LIN {X 0,Y 573.239,Z 232.081,A -85,B 0,C 180,E1 -2291.594,E2 -2291.594} C_VEL
LIN {X 0,Y 573.228,Z 232.079,A -85,B 0,C 180,E1 -2294.334,E2 -2294.334} C_VEL
LIN {X 0,Y 573.226,Z 232.083,A -85,B 0,C 180,E1 -2297.36,E2 -2297.36} C_VEL
LIN {X 0,Y 573.227,Z 232.083,A -85,B 0,C 180,E1 -2300.391,E2 -2300.391} C_VEL
LIN {X 0,Y 573.23,Z 232.078,A -85,B 0,C 180,E1 -2303.076,E2 -2303.076} C_VEL
LIN {X 0,Y 573.267,Z 232.08,A -85,B 0,C 180,E1 -2305.671,E2 -2305.671} C_VEL
LIN {X 0,Y 573.251,Z 232.076,A -85,B 0,C 180,E1 -2308.185,E2 -2308.185} C_VEL
LIN {X 0,Y 573.258,Z 232.079,A -85,B 0,C 180,E1 -2310.634,E2 -2310.634} C_VEL
LIN {X 0,Y 573.212,Z 232.08,A -85,B 0,C 180,E1 -2313.513,E2 -2313.513} C_VEL
LIN {X 0,Y 573.208,Z 232.086,A -85,B 0,C 180,E1 -2316.133,E2 -2316.133} C_VEL
LIN {X 0,Y 573.254,Z 232.075,A -85,B 0,C 180,E1 -2318.709,E2 -2318.709} C_VEL
LIN {X 0,Y 573.225,Z 232.083,A -85,B 0,C 180,E1 -2321.411,E2 -2321.411} C_VEL
LIN {X 0,Y 573.244,Z 232.077,A -85,B 0,C 180,E1 -2323.621,E2 -2323.621} C_VEL
LIN {X 0,Y 573.259,Z 232.076,A -85,B 0,C 180,E1 -2325.807,E2 -2325.807} C_VEL
LIN {X 0,Y 573.265,Z 232.074,A -85,B 0,C 180,E1 -2328.746,E2 -2328.746} C_VEL
LIN {X 0,Y 573.243,Z 232.082,A -85,B 0,C 180,E1 -2331.54,E2 -2331.54} C_VEL
LIN {X 0,Y 573.238,Z 232.078,A -85,B 0,C 180,E1 -2333.665,E2 -2333.665} C_VEL
LIN {X 0,Y 573.226,Z 232.079,A -85,B 0,C 180,E1 -2335.781,E2 -2335.781} C_VEL
LIN {X 0,Y 573.311,Z 232.071,A -85,B 0,C 180,E1 -2337.892,E2 -2337.892} C_VEL
LIN {X 0,Y 573.318,Z 232.068,A -85,B 0,C 180,E1 -2340.702,E2 -2340.702} C_VEL
LIN {X 0,Y 573.216,Z 232.086,A -85,B 0,C 180,E1 -2343.515,E2 -2343.515} C_VEL
LIN {X 0,Y 573.281,Z 232.073,A -85,B 0,C 180,E1 -2345.628,E2 -2345.628} C_VEL
LIN {X 0,Y 573.269,Z 232.073,A -85,B 0,C 180,E1 -2347.75,E2 -2347.75} C_VEL
LIN {X 0,Y 573.267,Z 232.077,A -85,B 0,C 180,E1 -2350.597,E2 -2350.597} C_VEL
LIN {X 0,Y 573.264,Z 232.074,A -85,B 0,C 180,E1 -2352.749,E2 -2352.749} C_VEL
LIN {X 0,Y 573.227,Z 232.08,A -85,B 0,C 180,E1 -2354.92,E2 -2354.92} C_VEL
LIN {X 0,Y 573.216,Z 232.08,A -85,B 0,C 180,E1 -2357.85,E2 -2357.85} C_VEL
LIN {X 0,Y 573.238,Z 232.078,A -85,B 0,C 180,E1 -2360.077,E2 -2360.077} C_VEL
LIN {X 0,Y 573.236,Z 232.084,A -85,B 0,C 180,E1 -2362.338,E2 -2362.338} C_VEL
LIN {X 0,Y 573.25,Z 232.076,A -85,B 0,C 180,E1 -2364.37,E2 -2364.37} C_VEL
LIN {X 0,Y 572.626,Z 232.154,A -85,B 0,C 180,E1 -2364.956,E2 -2364.956} C_VEL
LIN {X 0,Y 569.79,Z 232.514,A -85,B 0,C 180,E1 -2365.907,E2 -2365.907} C_VEL
LIN {X 0,Y 567.357,Z 232.819,A -85,B 0,C 180,E1 -2366.673,E2 -2366.673} C_VEL
LIN {X 0,Y 566.295,Z 232.949,A -85,B 0,C 180,E1 -2367.264,E2 -2367.264} C_VEL
LIN {X 0,Y 566.201,Z 232.958,A -85,B 0,C 180,E1 -2367.464,E2 -2367.464} C_VEL
LIN {X 0,Y 566.165,Z 232.959,A -85,B 0,C 180,E1 -2369.771,E2 -2369.771} C_VEL
LIN {X 0,Y 566.201,Z 232.96,A -85,B 0,C 180,E1 -2372.429,E2 -2372.429} C_VEL
LIN {X 0,Y 566.171,Z 232.957,A -85,B 0,C 180,E1 -2374.988,E2 -2374.988} C_VEL
LIN {X 0,Y 566.194,Z 232.958,A -85,B 0,C 180,E1 -2377.461,E2 -2377.461} C_VEL
LIN {X 0,Y 566.209,Z 232.953,A -85,B 0,C 180,E1 -2380.199,E2 -2380.199} C_VEL
LIN {X 0,Y 566.19,Z 232.96,A -85,B 0,C 180,E1 -2383.056,E2 -2383.056} C_VEL
LIN {X 0,Y 566.147,Z 232.965,A -85,B 0,C 180,E1 -2386.055,E2 -2386.055} C_VEL
LIN {X 0,Y 566.158,Z 232.959,A -85,B 0,C 180,E1 -2388.859,E2 -2388.859} C_VEL
LIN {X 0,Y 566.212,Z 232.959,A -85,B 0,C 180,E1 -2391.442,E2 -2391.442} C_VEL
LIN {X 0,Y 566.142,Z 232.963,A -85,B 0,C 180,E1 -2394.306,E2 -2394.306} C_VEL
LIN {X 0,Y 566.181,Z 233.754,A -85,B 0,C 180,E1 -2395.18,E2 -2395.18} C_VEL
LIN {X 0,Y 566.128,Z 237.923,A -85,B 0,C 180,E1 -2397.737,E2 -2397.737} C_VEL
LIN {X 0,Y 566.072,Z 242.199,A -85,B 0,C 180,E1 -2400.352,E2 -2400.352} C_VEL
LIN {X 0,Y 566.044,Z 246.038,A -85,B 0,C 180,E1 -2402.652,E2 -2402.652} C_VEL
LIN {X 0,Y 566.044,Z 250.095,A -85,B 0,C 180,E1 -2405.03,E2 -2405.03} C_VEL
LIN {X 0,Y 565.985,Z 254.135,A -85,B 0,C 180,E1 -2407.36,E2 -2407.36} C_VEL
LIN {X 0,Y 565.954,Z 258.174,A -85,B 0,C 180,E1 -2409.653,E2 -2409.653} C_VEL
LIN {X 0,Y 565.908,Z 262.249,A -85,B 0,C 180,E1 -2411.912,E2 -2411.912} C_VEL
LIN {X 0,Y 565.89,Z 266.396,A -85,B 0,C 180,E1 -2414.144,E2 -2414.144} C_VEL
LIN {X 0,Y 565.905,Z 270.544,A -85,B 0,C 180,E1 -2416.352,E2 -2416.352} C_VEL
LIN {X 0,Y 565.903,Z 272.531,A -85,B 0,C 180,E1 -2417.402,E2 -2417.402} C_VEL
LIN {X 0,Y 566.906,Z 280.366,A -85,B 0,C 180,E1 -2417.607,E2 -2417.607} C_VEL
LIN {X 0,Y 566.754,Z 293.781,A -85,B 0,C 180,E1 -2418.012,E2 -2418.012} C_VEL
LIN {X 0,Y 566.661,Z 306.298,A -85,B 0,C 180,E1 -2418.554,E2 -2418.554} C_VEL
LIN {X 0,Y 566.529,Z 317.551,A -85,B 0,C 180,E1 -2419.191,E2 -2419.191} C_VEL
LIN {X 0,Y 566.337,Z 328.843,A -85,B 0,C 180,E1 -2419.995,E2 -2419.995} C_VEL
LIN {X 0,Y 566.238,Z 338.89,A -85,B 0,C 180,E1 -2420.895,E2 -2420.895} C_VEL
LIN {X 0,Y 566.113,Z 348.591,A -85,B 0,C 180,E1 -2421.972,E2 -2421.972} C_VEL
LIN {X 0,Y 566.05,Z 355.159,A -85,B 0,C 180,E1 -2422.868,E2 -2422.868} C_VEL
LIN {X 0,Y 566.003,Z 361.628,A -85,B 0,C 180,E1 -2423.942,E2 -2423.942} C_VEL
LIN {X 0,Y 565.878,Z 366.765,A -85,B 0,C 180,E1 -2425.013,E2 -2425.013} C_VEL
LIN {X 0,Y 565.926,Z 370.754,A -85,B 0,C 180,E1 -2426.084,E2 -2426.084} C_VEL
LIN {X 0,Y 565.878,Z 373.702,A -85,B 0,C 180,E1 -2427.153,E2 -2427.153} C_VEL
LIN {X 0,Y 565.839,Z 375.128,A -85,B 0,C 180,E1 -2427.865,E2 -2427.865} C_VEL
LIN {X 0,Y 565.841,Z 376.756,A -85,B 0,C 180,E1 -2429.288,E2 -2429.288} C_VEL
LIN {X 0,Y 565.839,Z 376.996,A -85,B 0,C 180,E1 -2430,E2 -2430} C_VEL
LIN {X 0,Y 565.841,Z 376.815,A -85,B 0,C 180,E1 -2430.712,E2 -2430.712} C_VEL
LIN {X 0,Y 565.838,Z 375.268,A -85,B 0,C 180,E1 -2432.136,E2 -2432.136} C_VEL
LIN {X 0,Y 565.879,Z 373.907,A -85,B 0,C 180,E1 -2432.848,E2 -2432.848} C_VEL
LIN {X 0,Y 565.926,Z 371.029,A -85,B 0,C 180,E1 -2433.917,E2 -2433.917} C_VEL
LIN {X 0,Y 565.878,Z 367.129,A -85,B 0,C 180,E1 -2434.988,E2 -2434.988} C_VEL
LIN {X 0,Y 565.99,Z 362.096,A -85,B 0,C 180,E1 -2436.059,E2 -2436.059} C_VEL
LIN {X 0,Y 566.031,Z 355.771,A -85,B 0,C 180,E1 -2437.133,E2 -2437.133} C_VEL
LIN {X 0,Y 566.128,Z 347.849,A -85,B 0,C 180,E1 -2438.208,E2 -2438.208} C_VEL
LIN {X 0,Y 566.249,Z 337.997,A -85,B 0,C 180,E1 -2439.285,E2 -2439.285} C_VEL
LIN {X 0,Y 566.405,Z 327.678,A -85,B 0,C 180,E1 -2440.184,E2 -2440.184} C_VEL
LIN {X 0,Y 566.502,Z 316.393,A -85,B 0,C 180,E1 -2440.973,E2 -2440.973} C_VEL
LIN {X 0,Y 566.692,Z 305.185,A -85,B 0,C 180,E1 -2441.592,E2 -2441.592} C_VEL
LIN {X 0,Y 566.791,Z 292.591,A -85,B 0,C 180,E1 -2442.119,E2 -2442.119} C_VEL
LIN {X 0,Y 566.935,Z 279.413,A -85,B 0,C 180,E1 -2442.507,E2 -2442.507} C_VEL
LIN {X 0,Y 565.906,Z 272.529,A -85,B 0,C 180,E1 -2442.689,E2 -2442.689} C_VEL
LIN {X 0,Y 565.918,Z 267.947,A -85,B 0,C 180,E1 -2445.117,E2 -2445.117} C_VEL
LIN {X 0,Y 565.923,Z 263.798,A -85,B 0,C 180,E1 -2447.341,E2 -2447.341} C_VEL
LIN {X 0,Y 565.942,Z 259.671,A -85,B 0,C 180,E1 -2449.59,E2 -2449.59} C_VEL
LIN {X 0,Y 565.983,Z 255.624,A -85,B 0,C 180,E1 -2451.871,E2 -2451.871} C_VEL
LIN {X 0,Y 565.981,Z 251.584,A -85,B 0,C 180,E1 -2454.191,E2 -2454.191} C_VEL
LIN {X 0,Y 566.025,Z 247.439,A -85,B 0,C 180,E1 -2456.622,E2 -2456.622} C_VEL
LIN {X 0,Y 566.094,Z 243.487,A -85,B 0,C 180,E1 -2458.959,E2 -2458.959} C_VEL
LIN {X 0,Y 566.094,Z 239.426,A -85,B 0,C 180,E1 -2461.428,E2 -2461.428} C_VEL
LIN {X 0,Y 566.153,Z 235.297,A -85,B 0,C 180,E1 -2463.96,E2 -2463.96} C_VEL
LIN {X 0,Y 566.16,Z 233.635,A -85,B 0,C 180,E1 -2464.986,E2 -2464.986} C_VEL
LIN {X 0,Y 566.143,Z 232.963,A -85,B 0,C 180,E1 -2465.694,E2 -2465.694} C_VEL
LIN {X 0,Y 566.214,Z 232.958,A -85,B 0,C 180,E1 -2468.558,E2 -2468.558} C_VEL
LIN {X 0,Y 566.168,Z 232.958,A -85,B 0,C 180,E1 -2471.14,E2 -2471.14} C_VEL
LIN {X 0,Y 566.149,Z 232.965,A -85,B 0,C 180,E1 -2474.041,E2 -2474.041} C_VEL
LIN {X 0,Y 566.196,Z 232.96,A -85,B 0,C 180,E1 -2477.084,E2 -2477.084} C_VEL
LIN {X 0,Y 566.217,Z 232.955,A -85,B 0,C 180,E1 -2480.314,E2 -2480.314} C_VEL
LIN {X 0,Y 566.203,Z 232.953,A -85,B 0,C 180,E1 -2483.43,E2 -2483.43} C_VEL
LIN {X 0,Y 566.199,Z 232.956,A -85,B 0,C 180,E1 -2486.268,E2 -2486.268} C_VEL
LIN {X 0,Y 566.183,Z 232.96,A -85,B 0,C 180,E1 -2488.926,E2 -2488.926} C_VEL
LIN {X 0,Y 566.196,Z 232.955,A -85,B 0,C 180,E1 -2491.856,E2 -2491.856} C_VEL
LIN {X 0,Y 566.218,Z 232.958,A -85,B 0,C 180,E1 -2494.251,E2 -2494.251} C_VEL
LIN {X 0,Y 566.173,Z 232.958,A -85,B 0,C 180,E1 -2496.719,E2 -2496.719} C_VEL
LIN {X 0,Y 566.208,Z 232.958,A -85,B 0,C 180,E1 -2499.663,E2 -2499.663} C_VEL
LIN {X 0,Y 566.174,Z 232.957,A -85,B 0,C 180,E1 -2501.921,E2 -2501.921} C_VEL
LIN {X 0,Y 566.188,Z 232.96,A -85,B 0,C 180,E1 -2504.89,E2 -2504.89} C_VEL
LIN {X 0,Y 566.241,Z 232.953,A -85,B 0,C 180,E1 -2507.819,E2 -2507.819} C_VEL
LIN {X 0,Y 566.212,Z 232.953,A -85,B 0,C 180,E1 -2510.714,E2 -2510.714} C_VEL
LIN {X 0,Y 566.22,Z 232.958,A -85,B 0,C 180,E1 -2513.205,E2 -2513.205} C_VEL
LIN {X 0,Y 566.265,Z 232.952,A -85,B 0,C 180,E1 -2515.016,E2 -2515.016} C_VEL
LIN {X 0,Y 566.264,Z 232.948,A -85,B 0,C 180,E1 -2517.866,E2 -2517.866} C_VEL
LIN {X 0,Y 566.301,Z 232.942,A -85,B 0,C 180,E1 -2520.711,E2 -2520.711} C_VEL
LIN {X 0,Y 566.275,Z 232.946,A -85,B 0,C 180,E1 -2522.846,E2 -2522.846} C_VEL
LIN {X 0,Y 566.258,Z 232.948,A -85,B 0,C 180,E1 -2525.698,E2 -2525.698} C_VEL
LIN {X 0,Y 566.197,Z 232.961,A -85,B 0,C 180,E1 -2528.566,E2 -2528.566} C_VEL
LIN {X 0,Y 566.197,Z 232.955,A -85,B 0,C 180,E1 -2531.455,E2 -2531.455} C_VEL
LIN {X 0,Y 566.226,Z 232.951,A -85,B 0,C 180,E1 -2534.501,E2 -2534.501} C_VEL
LIN {X 0,Y 566.203,Z 232.959,A -85,B 0,C 180,E1 -2537.332,E2 -2537.332} C_VEL
LIN {X 0,Y 566.211,Z 232.957,A -85,B 0,C 180,E1 -2540.337,E2 -2540.337} C_VEL
LIN {X 0,Y 566.168,Z 232.958,A -85,B 0,C 180,E1 -2543.28,E2 -2543.28} C_VEL
LIN {X 0,Y 566.189,Z 232.963,A -85,B 0,C 180,E1 -2545.75,E2 -2545.75} C_VEL
LIN {X 0,Y 566.188,Z 232.956,A -85,B 0,C 180,E1 -2548.198,E2 -2548.198} C_VEL
LIN {X 0,Y 566.192,Z 232.96,A -85,B 0,C 180,E1 -2551.076,E2 -2551.076} C_VEL
LIN {X 0,Y 566.215,Z 232.953,A -85,B 0,C 180,E1 -2553.734,E2 -2553.734} C_VEL
LIN {X 0,Y 566.183,Z 232.957,A -85,B 0,C 180,E1 -2556.571,E2 -2556.571} C_VEL
LIN {X 0,Y 566.206,Z 232.957,A -85,B 0,C 180,E1 -2559.684,E2 -2559.684} C_VEL
LIN {X 0,Y 566.175,Z 232.957,A -85,B 0,C 180,E1 -2562.091,E2 -2562.091} C_VEL
LIN {X 0,Y 566.167,Z 232.96,A -85,B 0,C 180,E1 -2565.037,E2 -2565.037} C_VEL
LIN {X 0,Y 566.192,Z 232.962,A -85,B 0,C 180,E1 -2567.91,E2 -2567.91} C_VEL
LIN {X 0,Y 566.212,Z 232.954,A -85,B 0,C 180,E1 -2570.726,E2 -2570.726} C_VEL
LIN {X 0,Y 566.222,Z 233.113,A -85,B 0,C 180,E1 -2573.638,E2 -2573.638} C_VEL
LIN {X 0,Y 566.512,Z 236.983,A -85,B 0,C 180,E1 -2575.203,E2 -2575.203} C_VEL
LIN {X 0,Y 566.453,Z 243.602,A -85,B 0,C 180,E1 -2577.757,E2 -2577.757} C_VEL
LIN {X 0,Y 566.335,Z 251.568,A -85,B 0,C 180,E1 -2580.68,E2 -2580.68} C_VEL
LIN {X 0,Y 566.252,Z 259.349,A -85,B 0,C 180,E1 -2583.46,E2 -2583.46} C_VEL
LIN {X 0,Y 566.223,Z 267.275,A -85,B 0,C 180,E1 -2586.209,E2 -2586.209} C_VEL
LIN {X 0,Y 566.155,Z 275.17,A -85,B 0,C 180,E1 -2588.9,E2 -2588.9} C_VEL
LIN {X 0,Y 566.088,Z 283.03,A -85,B 0,C 180,E1 -2591.543,E2 -2591.543} C_VEL
LIN {X 0,Y 566.028,Z 291.935,A -85,B 0,C 180,E1 -2594.517,E2 -2594.517} C_VEL
LIN {X 0,Y 565.98,Z 300.491,A -85,B 0,C 180,E1 -2597.335,E2 -2597.335} C_VEL
LIN {X 0,Y 566.952,Z 307.503,A -85,B 0,C 180,E1 -2597.494,E2 -2597.494} C_VEL
LIN {X 0,Y 566.827,Z 319.872,A -85,B 0,C 180,E1 -2597.832,E2 -2597.832} C_VEL
LIN {X 0,Y 566.645,Z 332.902,A -85,B 0,C 180,E1 -2598.346,E2 -2598.346} C_VEL
LIN {X 0,Y 566.526,Z 344.488,A -85,B 0,C 180,E1 -2598.955,E2 -2598.955} C_VEL
LIN {X 0,Y 566.438,Z 355.922,A -85,B 0,C 180,E1 -2599.726,E2 -2599.726} C_VEL
LIN {X 0,Y 566.282,Z 365.599,A -85,B 0,C 180,E1 -2600.535,E2 -2600.535} C_VEL
LIN {X 0,Y 566.181,Z 374.412,A -85,B 0,C 180,E1 -2601.433,E2 -2601.433} C_VEL
LIN {X 0,Y 566.056,Z 383.001,A -85,B 0,C 180,E1 -2602.509,E2 -2602.509} C_VEL
LIN {X 0,Y 565.965,Z 389.868,A -85,B 0,C 180,E1 -2603.583,E2 -2603.583} C_VEL
LIN {X 0,Y 565.937,Z 395.365,A -85,B 0,C 180,E1 -2604.656,E2 -2604.656} C_VEL
LIN {X 0,Y 565.959,Z 399.677,A -85,B 0,C 180,E1 -2605.727,E2 -2605.727} C_VEL
LIN {X 0,Y 565.927,Z 401.957,A -85,B 0,C 180,E1 -2606.44,E2 -2606.44} C_VEL
LIN {X 0,Y 565.878,Z 403.808,A -85,B 0,C 180,E1 -2607.152,E2 -2607.152} C_VEL
LIN {X 0,Y 565.846,Z 406.185,A -85,B 0,C 180,E1 -2608.577,E2 -2608.577} C_VEL
LIN {X 0,Y 565.839,Z 407,A -85,B 0,C 180,E1 -2610,E2 -2610} C_VEL
LIN {X 0,Y 565.846,Z 406.186,A -85,B 0,C 180,E1 -2611.423,E2 -2611.423} C_VEL
LIN {X 0,Y 565.878,Z 403.81,A -85,B 0,C 180,E1 -2612.847,E2 -2612.847} C_VEL
LIN {X 0,Y 565.926,Z 400.896,A -85,B 0,C 180,E1 -2613.916,E2 -2613.916} C_VEL
LIN {X 0,Y 565.878,Z 396.949,A -85,B 0,C 180,E1 -2614.987,E2 -2614.987} C_VEL
LIN {X 0,Y 566.002,Z 391.867,A -85,B 0,C 180,E1 -2616.058,E2 -2616.058} C_VEL
LIN {X 0,Y 566.04,Z 385.468,A -85,B 0,C 180,E1 -2617.132,E2 -2617.132} C_VEL
LIN {X 0,Y 566.134,Z 377.478,A -85,B 0,C 180,E1 -2618.208,E2 -2618.208} C_VEL
LIN {X 0,Y 566.229,Z 369.335,A -85,B 0,C 180,E1 -2619.105,E2 -2619.105} C_VEL
LIN {X 0,Y 566.339,Z 359.4,A -85,B 0,C 180,E1 -2620.005,E2 -2620.005} C_VEL
LIN {X 0,Y 566.471,Z 348.335,A -85,B 0,C 180,E1 -2620.806,E2 -2620.806} C_VEL
LIN {X 0,Y 566.608,Z 335.946,A -85,B 0,C 180,E1 -2621.51,E2 -2621.51} C_VEL
LIN {X 0,Y 566.742,Z 323.768,A -85,B 0,C 180,E1 -2622.034,E2 -2622.034} C_VEL
LIN {X 0,Y 566.913,Z 310.348,A -85,B 0,C 180,E1 -2622.439,E2 -2622.439} C_VEL
LIN {X 0,Y 566.643,Z 304.812,A -85,B 0,C 180,E1 -2622.567,E2 -2622.567} C_VEL
LIN {X 0,Y 565.98,Z 300.492,A -85,B 0,C 180,E1 -2622.665,E2 -2622.665} C_VEL
LIN {X 0,Y 566.028,Z 291.935,A -85,B 0,C 180,E1 -2625.483,E2 -2625.483} C_VEL
LIN {X 0,Y 566.088,Z 283.031,A -85,B 0,C 180,E1 -2628.456,E2 -2628.456} C_VEL
LIN {X 0,Y 566.201,Z 274.237,A -85,B 0,C 180,E1 -2631.417,E2 -2631.417} C_VEL
LIN {X 0,Y 566.213,Z 265.01,A -85,B 0,C 180,E1 -2634.57,E2 -2634.57} C_VEL
LIN {X 0,Y 566.242,Z 257.102,A -85,B 0,C 180,E1 -2637.338,E2 -2637.338} C_VEL
LIN {X 0,Y 566.351,Z 249.228,A -85,B 0,C 180,E1 -2640.171,E2 -2640.171} C_VEL
LIN {X 0,Y 566.478,Z 241.385,A -85,B 0,C 180,E1 -2643.085,E2 -2643.085} C_VEL
LIN {X 0,Y 566.479,Z 234.789,A -85,B 0,C 180,E1 -2645.669,E2 -2645.669} C_VEL
LIN {X 0,Y 566.205,Z 232.96,A -85,B 0,C 180,E1 -2646.466,E2 -2646.466} C_VEL
LIN {X 0,Y 566.213,Z 232.955,A -85,B 0,C 180,E1 -2649.685,E2 -2649.685} C_VEL
LIN {X 0,Y 566.211,Z 232.96,A -85,B 0,C 180,E1 -2652.088,E2 -2652.088} C_VEL
LIN {X 0,Y 566.17,Z 232.96,A -85,B 0,C 180,E1 -2655.036,E2 -2655.036} C_VEL
LIN {X 0,Y 566.174,Z 232.957,A -85,B 0,C 180,E1 -2657.909,E2 -2657.909} C_VEL
LIN {X 0,Y 566.203,Z 232.959,A -85,B 0,C 180,E1 -2660.725,E2 -2660.725} C_VEL
LIN {X 0,Y 566.182,Z 232.957,A -85,B 0,C 180,E1 -2663.429,E2 -2663.429} C_VEL
LIN {X 0,Y 566.214,Z 232.954,A -85,B 0,C 180,E1 -2666.266,E2 -2666.266} C_VEL
LIN {X 0,Y 566.196,Z 232.959,A -85,B 0,C 180,E1 -2668.923,E2 -2668.923} C_VEL
LIN {X 0,Y 566.189,Z 232.956,A -85,B 0,C 180,E1 -2671.856,E2 -2671.856} C_VEL
LIN {X 0,Y 566.189,Z 232.962,A -85,B 0,C 180,E1 -2674.25,E2 -2674.25} C_VEL
LIN {X 0,Y 566.178,Z 232.959,A -85,B 0,C 180,E1 -2677.368,E2 -2677.368} C_VEL
LIN {X 0,Y 566.21,Z 232.957,A -85,B 0,C 180,E1 -2679.663,E2 -2679.663} C_VEL
LIN {X 0,Y 566.202,Z 232.959,A -85,B 0,C 180,E1 -2682.668,E2 -2682.668} C_VEL
LIN {X 0,Y 566.222,Z 232.952,A -85,B 0,C 180,E1 -2685.626,E2 -2685.626} C_VEL
LIN {X 0,Y 566.236,Z 232.95,A -85,B 0,C 180,E1 -2688.676,E2 -2688.676} C_VEL
LIN {X 0,Y 566.195,Z 232.962,A -85,B 0,C 180,E1 -2691.434,E2 -2691.434} C_VEL
LIN {X 0,Y 566.203,Z 232.955,A -85,B 0,C 180,E1 -2693.586,E2 -2693.586} C_VEL
LIN {X 0,Y 566.184,Z 232.956,A -85,B 0,C 180,E1 -2695.729,E2 -2695.729} C_VEL
LIN {X 0,Y 566.283,Z 232.946,A -85,B 0,C 180,E1 -2697.866,E2 -2697.866} C_VEL
LIN {X 0,Y 566.29,Z 232.943,A -85,B 0,C 180,E1 -2700.711,E2 -2700.711} C_VEL
LIN {X 0,Y 566.25,Z 232.949,A -85,B 0,C 180,E1 -2702.846,E2 -2702.846} C_VEL
LIN {X 0,Y 566.247,Z 232.948,A -85,B 0,C 180,E1 -2705.698,E2 -2705.698} C_VEL
LIN {X 0,Y 566.209,Z 232.959,A -85,B 0,C 180,E1 -2708.566,E2 -2708.566} C_VEL
LIN {X 0,Y 566.245,Z 232.95,A -85,B 0,C 180,E1 -2711.454,E2 -2711.454} C_VEL
LIN {X 0,Y 566.221,Z 232.952,A -85,B 0,C 180,E1 -2714.5,E2 -2714.5} C_VEL
LIN {X 0,Y 566.188,Z 232.96,A -85,B 0,C 180,E1 -2717.332,E2 -2717.332} C_VEL
LIN {X 0,Y 566.202,Z 232.953,A -85,B 0,C 180,E1 -2719.581,E2 -2719.581} C_VEL
LIN {X 0,Y 566.195,Z 232.956,A -85,B 0,C 180,E1 -2721.863,E2 -2721.863} C_VEL
LIN {X 0,Y 566.221,Z 232.952,A -85,B 0,C 180,E1 -2725.03,E2 -2725.03} C_VEL
LIN {X 0,Y 566.201,Z 232.958,A -85,B 0,C 180,E1 -2727.464,E2 -2727.464} C_VEL
LIN {X 0,Y 565.509,Z 233.042,A -85,B 0,C 180,E1 -2728.058,E2 -2728.058} C_VEL
LIN {X 0,Y 562.635,Z 233.404,A -85,B 0,C 180,E1 -2729.021,E2 -2729.021} C_VEL
LIN {X 0,Y 560.226,Z 233.701,A -85,B 0,C 180,E1 -2729.797,E2 -2729.797} C_VEL
LIN {X 0,Y 559.203,Z 233.828,A -85,B 0,C 180,E1 -2730.395,E2 -2730.395} C_VEL
LIN {X 0,Y 559.125,Z 233.836,A -85,B 0,C 180,E1 -2730.598,E2 -2730.598} C_VEL
LIN {X 0,Y 559.151,Z 233.837,A -85,B 0,C 180,E1 -2732.716,E2 -2732.716} C_VEL
LIN {X 0,Y 559.12,Z 233.836,A -85,B 0,C 180,E1 -2735.325,E2 -2735.325} C_VEL
LIN {X 0,Y 559.132,Z 233.837,A -85,B 0,C 180,E1 -2738.018,E2 -2738.018} C_VEL
LIN {X 0,Y 559.158,Z 233.835,A -85,B 0,C 180,E1 -2740.813,E2 -2740.813} C_VEL
LIN {X 0,Y 559.112,Z 233.837,A -85,B 0,C 180,E1 -2743.737,E2 -2743.737} C_VEL
LIN {X 0,Y 559.095,Z 233.845,A -85,B 0,C 180,E1 -2746.261,E2 -2746.261} C_VEL
LIN {X 0,Y 559.12,Z 233.836,A -85,B 0,C 180,E1 -2748.955,E2 -2748.955} C_VEL
LIN {X 0,Y 559.176,Z 233.833,A -85,B 0,C 180,E1 -2751.192,E2 -2751.192} C_VEL
LIN {X 0,Y 559.124,Z 233.836,A -85,B 0,C 180,E1 -2753.788,E2 -2753.788} C_VEL
LIN {X 0,Y 559.096,Z 234.003,A -85,B 0,C 180,E1 -2754.793,E2 -2754.793} C_VEL
LIN {X 0,Y 559.064,Z 238.161,A -85,B 0,C 180,E1 -2757.38,E2 -2757.38} C_VEL
LIN {X 0,Y 559.031,Z 242.66,A -85,B 0,C 180,E1 -2760.164,E2 -2760.164} C_VEL
LIN {X 0,Y 558.985,Z 246.144,A -85,B 0,C 180,E1 -2762.277,E2 -2762.277} C_VEL
LIN {X 0,Y 558.938,Z 251.549,A -85,B 0,C 180,E1 -2765.485,E2 -2765.485} C_VEL
LIN {X 0,Y 558.923,Z 256.778,A -85,B 0,C 180,E1 -2768.512,E2 -2768.512} C_VEL
LIN {X 0,Y 558.881,Z 261.006,A -85,B 0,C 180,E1 -2770.916,E2 -2770.916} C_VEL
LIN {X 0,Y 558.859,Z 265.015,A -85,B 0,C 180,E1 -2773.188,E2 -2773.188} C_VEL
LIN {X 0,Y 558.818,Z 270.545,A -85,B 0,C 180,E1 -2776.175,E2 -2776.175} C_VEL
LIN {X 0,Y 558.836,Z 272.532,A -85,B 0,C 180,E1 -2777.24,E2 -2777.24} C_VEL
LIN {X 0,Y 559.969,Z 280.388,A -85,B 0,C 180,E1 -2777.45,E2 -2777.45} C_VEL
LIN {X 0,Y 559.824,Z 293.797,A -85,B 0,C 180,E1 -2777.862,E2 -2777.862} C_VEL
LIN {X 0,Y 559.687,Z 306.308,A -85,B 0,C 180,E1 -2778.41,E2 -2778.41} C_VEL
LIN {X 0,Y 559.539,Z 317.651,A -85,B 0,C 180,E1 -2779.06,E2 -2779.06} C_VEL
LIN {X 0,Y 559.349,Z 328.852,A -85,B 0,C 180,E1 -2779.869,E2 -2779.869} C_VEL
LIN {X 0,Y 559.21,Z 338.895,A -85,B 0,C 180,E1 -2780.779,E2 -2780.779} C_VEL
LIN {X 0,Y 559.05,Z 348.595,A -85,B 0,C 180,E1 -2781.87,E2 -2781.87} C_VEL
LIN {X 0,Y 558.971,Z 356.456,A -85,B 0,C 180,E1 -2782.977,E2 -2782.977} C_VEL
LIN {X 0,Y 558.936,Z 363.454,A -85,B 0,C 180,E1 -2784.227,E2 -2784.227} C_VEL
LIN {X 0,Y 558.826,Z 368.195,A -85,B 0,C 180,E1 -2785.311,E2 -2785.311} C_VEL
LIN {X 0,Y 558.836,Z 371.828,A -85,B 0,C 180,E1 -2786.395,E2 -2786.395} C_VEL
LIN {X 0,Y 558.799,Z 373.704,A -85,B 0,C 180,E1 -2787.116,E2 -2787.116} C_VEL
LIN {X 0,Y 558.745,Z 375.128,A -85,B 0,C 180,E1 -2787.838,E2 -2787.838} C_VEL
LIN {X 0,Y 558.741,Z 376.757,A -85,B 0,C 180,E1 -2789.279,E2 -2789.279} C_VEL
LIN {X 0,Y 558.74,Z 376.996,A -85,B 0,C 180,E1 -2790,E2 -2790} C_VEL
LIN {X 0,Y 558.741,Z 376.815,A -85,B 0,C 180,E1 -2790.721,E2 -2790.721} C_VEL
LIN {X 0,Y 558.745,Z 375.266,A -85,B 0,C 180,E1 -2792.163,E2 -2792.163} C_VEL
LIN {X 0,Y 558.8,Z 373.905,A -85,B 0,C 180,E1 -2792.884,E2 -2792.884} C_VEL
LIN {X 0,Y 558.844,Z 371.027,A -85,B 0,C 180,E1 -2793.966,E2 -2793.966} C_VEL
LIN {X 0,Y 558.798,Z 367.126,A -85,B 0,C 180,E1 -2795.051,E2 -2795.051} C_VEL
LIN {X 0,Y 558.91,Z 362.094,A -85,B 0,C 180,E1 -2796.136,E2 -2796.136} C_VEL
LIN {X 0,Y 558.973,Z 355.767,A -85,B 0,C 180,E1 -2797.223,E2 -2797.223} C_VEL
LIN {X 0,Y 559.091,Z 347.844,A -85,B 0,C 180,E1 -2798.312,E2 -2798.312} C_VEL
LIN {X 0,Y 559.223,Z 337.991,A -85,B 0,C 180,E1 -2799.403,E2 -2799.403} C_VEL
LIN {X 0,Y 559.399,Z 327.671,A -85,B 0,C 180,E1 -2800.313,E2 -2800.313} C_VEL
LIN {X 0,Y 559.519,Z 316.7,A -85,B 0,C 180,E1 -2801.092,E2 -2801.092} C_VEL
LIN {X 0,Y 559.73,Z 305.173,A -85,B 0,C 180,E1 -2801.738,E2 -2801.738} C_VEL
LIN {X 0,Y 559.849,Z 292.574,A -85,B 0,C 180,E1 -2802.272,E2 -2802.272} C_VEL
LIN {X 0,Y 559.933,Z 279.389,A -85,B 0,C 180,E1 -2802.666,E2 -2802.666} C_VEL
LIN {X 0,Y 558.805,Z 272.528,A -85,B 0,C 180,E1 -2802.853,E2 -2802.853} C_VEL
LIN {X 0,Y 558.832,Z 267.946,A -85,B 0,C 180,E1 -2805.314,E2 -2805.314} C_VEL
LIN {X 0,Y 558.839,Z 263.829,A -85,B 0,C 180,E1 -2807.567,E2 -2807.567} C_VEL
LIN {X 0,Y 558.876,Z 259.827,A -85,B 0,C 180,E1 -2809.848,E2 -2809.848} C_VEL
LIN {X 0,Y 558.924,Z 255.746,A -85,B 0,C 180,E1 -2812.162,E2 -2812.162} C_VEL
LIN {X 0,Y 558.969,Z 250.345,A -85,B 0,C 180,E1 -2815.308,E2 -2815.308} C_VEL
LIN {X 0,Y 559.034,Z 244.942,A -85,B 0,C 180,E1 -2818.537,E2 -2818.537} C_VEL
LIN {X 0,Y 559.058,Z 240.5,A -85,B 0,C 180,E1 -2821.258,E2 -2821.258} C_VEL
LIN {X 0,Y 559.107,Z 235.36,A -85,B 0,C 180,E1 -2824.448,E2 -2824.448} C_VEL
LIN {X 0,Y 559.09,Z 233.956,A -85,B 0,C 180,E1 -2825.327,E2 -2825.327} C_VEL
LIN {X 0,Y 559.136,Z 233.834,A -85,B 0,C 180,E1 -2828.018,E2 -2828.018} C_VEL
LIN {X 0,Y 559.156,Z 233.833,A -85,B 0,C 180,E1 -2830.813,E2 -2830.813} C_VEL
LIN {X 0,Y 559.096,Z 233.844,A -85,B 0,C 180,E1 -2833.739,E2 -2833.739} C_VEL
LIN {X 0,Y 559.112,Z 233.838,A -85,B 0,C 180,E1 -2836.263,E2 -2836.263} C_VEL
LIN {X 0,Y 559.159,Z 233.836,A -85,B 0,C 180,E1 -2839.188,E2 -2839.188} C_VEL
LIN {X 0,Y 559.135,Z 233.836,A -85,B 0,C 180,E1 -2841.982,E2 -2841.982} C_VEL
LIN {X 0,Y 559.133,Z 233.834,A -85,B 0,C 180,E1 -2844.787,E2 -2844.787} C_VEL
LIN {X 0,Y 559.155,Z 233.836,A -85,B 0,C 180,E1 -2847.365,E2 -2847.365} C_VEL
LIN {X 0,Y 559.115,Z 233.837,A -85,B 0,C 180,E1 -2850.149,E2 -2850.149} C_VEL
LIN {X 0,Y 559.174,Z 233.831,A -85,B 0,C 180,E1 -2853.173,E2 -2853.173} C_VEL
LIN {X 0,Y 559.16,Z 233.832,A -85,B 0,C 180,E1 -2855.495,E2 -2855.495} C_VEL
LIN {X 0,Y 559.176,Z 233.828,A -85,B 0,C 180,E1 -2858.624,E2 -2858.624} C_VEL
LIN {X 0,Y 559.161,Z 233.834,A -85,B 0,C 180,E1 -2860.926,E2 -2860.926} C_VEL
LIN {X 0,Y 559.141,Z 233.834,A -85,B 0,C 180,E1 -2863.947,E2 -2863.947} C_VEL
LIN {X 0,Y 559.162,Z 233.836,A -85,B 0,C 180,E1 -2866.184,E2 -2866.184} C_VEL
LIN {X 0,Y 559.197,Z 233.827,A -85,B 0,C 180,E1 -2869.133,E2 -2869.133} C_VEL
LIN {X 0,Y 559.195,Z 233.827,A -85,B 0,C 180,E1 -2872.053,E2 -2872.053} C_VEL
LIN {X 0,Y 559.241,Z 233.828,A -85,B 0,C 180,E1 -2874.953,E2 -2874.953} C_VEL
LIN {X 0,Y 559.237,Z 233.823,A -85,B 0,C 180,E1 -2877.839,E2 -2877.839} C_VEL
LIN {X 0,Y 559.272,Z 233.818,A -85,B 0,C 180,E1 -2880.72,E2 -2880.72} C_VEL
LIN {X 0,Y 559.241,Z 233.822,A -85,B 0,C 180,E1 -2882.881,E2 -2882.881} C_VEL
LIN {X 0,Y 559.227,Z 233.824,A -85,B 0,C 180,E1 -2885.77,E2 -2885.77} C_VEL
LIN {X 0,Y 559.162,Z 233.837,A -85,B 0,C 180,E1 -2888.675,E2 -2888.675} C_VEL
LIN {X 0,Y 559.163,Z 233.832,A -85,B 0,C 180,E1 -2891.601,E2 -2891.601} C_VEL
LIN {X 0,Y 559.184,Z 233.828,A -85,B 0,C 180,E1 -2894.588,E2 -2894.588} C_VEL
LIN {X 0,Y 559.162,Z 233.834,A -85,B 0,C 180,E1 -2897.557,E2 -2897.557} C_VEL
LIN {X 0,Y 559.17,Z 233.83,A -85,B 0,C 180,E1 -2899.838,E2 -2899.838} C_VEL
LIN {X 0,Y 559.142,Z 233.838,A -85,B 0,C 180,E1 -2902.153,E2 -2902.153} C_VEL
LIN {X 0,Y 559.141,Z 233.834,A -85,B 0,C 180,E1 -2905.178,E2 -2905.178} C_VEL
LIN {X 0,Y 559.129,Z 233.839,A -85,B 0,C 180,E1 -2907.715,E2 -2907.715} C_VEL
LIN {X 0,Y 559.142,Z 233.834,A -85,B 0,C 180,E1 -2910.184,E2 -2910.184} C_VEL
LIN {X 0,Y 559.161,Z 233.837,A -85,B 0,C 180,E1 -2912.715,E2 -2912.715} C_VEL
LIN {X 0,Y 559.126,Z 233.836,A -85,B 0,C 180,E1 -2915.324,E2 -2915.324} C_VEL
LIN {X 0,Y 559.125,Z 233.838,A -85,B 0,C 180,E1 -2918.018,E2 -2918.018} C_VEL
LIN {X 0,Y 559.155,Z 233.834,A -85,B 0,C 180,E1 -2920.813,E2 -2920.813} C_VEL
LIN {X 0,Y 559.138,Z 233.834,A -85,B 0,C 180,E1 -2923.734,E2 -2923.734} C_VEL
LIN {X 0,Y 559.148,Z 233.834,A -85,B 0,C 180,E1 -2926.804,E2 -2926.804} C_VEL
LIN {X 0,Y 559.158,Z 233.833,A -85,B 0,C 180,E1 -2929.188,E2 -2929.188} C_VEL
LIN {X 0,Y 559.13,Z 233.838,A -85,B 0,C 180,E1 -2931.982,E2 -2931.982} C_VEL
LIN {X 0,Y 559.189,Z 233.886,A -85,B 0,C 180,E1 -2933.438,E2 -2933.438} C_VEL
LIN {X 0,Y 559.515,Z 238.065,A -85,B 0,C 180,E1 -2935.155,E2 -2935.155} C_VEL
LIN {X 0,Y 559.434,Z 244.655,A -85,B 0,C 180,E1 -2937.735,E2 -2937.735} C_VEL
LIN {X 0,Y 559.32,Z 252.511,A -85,B 0,C 180,E1 -2940.656,E2 -2940.656} C_VEL
LIN {X 0,Y 559.204,Z 260.468,A -85,B 0,C 180,E1 -2943.534,E2 -2943.534} C_VEL
LIN {X 0,Y 559.173,Z 268.31,A -85,B 0,C 180,E1 -2946.284,E2 -2946.284} C_VEL
LIN {X 0,Y 559.1,Z 276.181,A -85,B 0,C 180,E1 -2949.007,E2 -2949.007} C_VEL
LIN {X 0,Y 559.019,Z 284.123,A -85,B 0,C 180,E1 -2951.681,E2 -2951.681} C_VEL
LIN {X 0,Y 558.965,Z 291.935,A -85,B 0,C 180,E1 -2954.316,E2 -2954.316} C_VEL
LIN {X 0,Y 558.922,Z 300.491,A -85,B 0,C 180,E1 -2957.173,E2 -2957.173} C_VEL
LIN {X 0,Y 560.013,Z 308.516,A -85,B 0,C 180,E1 -2957.359,E2 -2957.359} C_VEL
LIN {X 0,Y 559.877,Z 321.301,A -85,B 0,C 180,E1 -2957.729,E2 -2957.729} C_VEL
LIN {X 0,Y 559.695,Z 332.277,A -85,B 0,C 180,E1 -2958.17,E2 -2958.17} C_VEL
LIN {X 0,Y 559.538,Z 343.913,A -85,B 0,C 180,E1 -2958.781,E2 -2958.781} C_VEL
LIN {X 0,Y 559.433,Z 354.743,A -85,B 0,C 180,E1 -2959.504,E2 -2959.504} C_VEL
LIN {X 0,Y 559.243,Z 365.598,A -85,B 0,C 180,E1 -2960.415,E2 -2960.415} C_VEL
LIN {X 0,Y 559.127,Z 374.412,A -85,B 0,C 180,E1 -2961.325,E2 -2961.325} C_VEL
LIN {X 0,Y 558.996,Z 383.002,A -85,B 0,C 180,E1 -2962.414,E2 -2962.414} C_VEL
LIN {X 0,Y 558.885,Z 390.687,A -85,B 0,C 180,E1 -2963.649,E2 -2963.649} C_VEL
LIN {X 0,Y 558.869,Z 395.365,A -85,B 0,C 180,E1 -2964.588,E2 -2964.588} C_VEL
LIN {X 0,Y 558.869,Z 399.677,A -85,B 0,C 180,E1 -2965.673,E2 -2965.673} C_VEL
LIN {X 0,Y 558.836,Z 401.958,A -85,B 0,C 180,E1 -2966.395,E2 -2966.395} C_VEL
LIN {X 0,Y 558.799,Z 403.807,A -85,B 0,C 180,E1 -2967.116,E2 -2967.116} C_VEL
LIN {X 0,Y 558.745,Z 406.184,A -85,B 0,C 180,E1 -2968.558,E2 -2968.558} C_VEL
LIN {X 0,Y 558.74,Z 407,A -85,B 0,C 180,E1 -2970,E2 -2970} C_VEL
LIN {X 0,Y 558.745,Z 406.185,A -85,B 0,C 180,E1 -2971.441,E2 -2971.441} C_VEL
LIN {X 0,Y 558.799,Z 403.81,A -85,B 0,C 180,E1 -2972.884,E2 -2972.884} C_VEL
LIN {X 0,Y 558.844,Z 400.896,A -85,B 0,C 180,E1 -2973.966,E2 -2973.966} C_VEL
LIN {X 0,Y 558.798,Z 396.949,A -85,B 0,C 180,E1 -2975.051,E2 -2975.051} C_VEL
LIN {X 0,Y 558.922,Z 391.867,A -85,B 0,C 180,E1 -2976.135,E2 -2976.135} C_VEL
LIN {X 0,Y 558.977,Z 385.468,A -85,B 0,C 180,E1 -2977.223,E2 -2977.223} C_VEL
LIN {X 0,Y 559.099,Z 377.478,A -85,B 0,C 180,E1 -2978.312,E2 -2978.312} C_VEL
LIN {X 0,Y 559.195,Z 369.335,A -85,B 0,C 180,E1 -2979.221,E2 -2979.221} C_VEL
LIN {X 0,Y 559.354,Z 359.399,A -85,B 0,C 180,E1 -2980.131,E2 -2980.131} C_VEL
LIN {X 0,Y 559.475,Z 348.444,A -85,B 0,C 180,E1 -2980.935,E2 -2980.935} C_VEL
LIN {X 0,Y 559.636,Z 336.817,A -85,B 0,C 180,E1 -2981.61,E2 -2981.61} C_VEL
LIN {X 0,Y 559.76,Z 324.98,A -85,B 0,C 180,E1 -2982.14,E2 -2982.14} C_VEL
LIN {X 0,Y 559.956,Z 312.175,A -85,B 0,C 180,E1 -2982.55,E2 -2982.55} C_VEL
LIN {X 0,Y 559.763,Z 305.951,A -85,B 0,C 180,E1 -2982.701,E2 -2982.701} C_VEL
LIN {X 0,Y 558.922,Z 300.492,A -85,B 0,C 180,E1 -2982.827,E2 -2982.827} C_VEL
LIN {X 0,Y 558.965,Z 291.935,A -85,B 0,C 180,E1 -2985.684,E2 -2985.684} C_VEL
LIN {X 0,Y 559.019,Z 284.124,A -85,B 0,C 180,E1 -2988.319,E2 -2988.319} C_VEL
LIN {X 0,Y 559.1,Z 276.182,A -85,B 0,C 180,E1 -2990.993,E2 -2990.993} C_VEL
LIN {X 0,Y 559.203,Z 267.179,A -85,B 0,C 180,E1 -2994.108,E2 -2994.108} C_VEL
LIN {X 0,Y 559.202,Z 259.257,A -85,B 0,C 180,E1 -2996.901,E2 -2996.901} C_VEL
LIN {X 0,Y 559.326,Z 251.029,A -85,B 0,C 180,E1 -2999.889,E2 -2999.889} C_VEL
LIN {X 0,Y 559.46,Z 243.528,A -85,B 0,C 180,E1 -3002.695,E2 -3002.695} C_VEL
LIN {X 0,Y 559.53,Z 236.932,A -85,B 0,C 180,E1 -3005.295,E2 -3005.295} C_VEL
LIN {X 0,Y 559.164,Z 233.838,A -85,B 0,C 180,E1 -3006.608,E2 -3006.608} C_VEL
LIN {X 0,Y 559.179,Z 233.833,A -85,B 0,C 180,E1 -3009.866,E2 -3009.866} C_VEL
LIN {X 0,Y 559.163,Z 233.831,A -85,B 0,C 180,E1 -3012.743,E2 -3012.743} C_VEL
LIN {X 0,Y 559.15,Z 233.835,A -85,B 0,C 180,E1 -3015.761,E2 -3015.761} C_VEL
LIN {X 0,Y 559.127,Z 233.836,A -85,B 0,C 180,E1 -3018.226,E2 -3018.226} C_VEL
LIN {X 0,Y 559.167,Z 233.83,A -85,B 0,C 180,E1 -3021.193,E2 -3021.193} C_VEL
LIN {X 0,Y 559.122,Z 233.84,A -85,B 0,C 180,E1 -3023.788,E2 -3023.788} C_VEL
LIN {X 0,Y 559.165,Z 233.831,A -85,B 0,C 180,E1 -3026.425,E2 -3026.425} C_VEL
LIN {X 0,Y 559.16,Z 233.837,A -85,B 0,C 180,E1 -3028.981,E2 -3028.981} C_VEL
LIN {X 0,Y 559.135,Z 233.834,A -85,B 0,C 180,E1 -3031.625,E2 -3031.625} C_VEL
LIN {X 0,Y 559.157,Z 233.833,A -85,B 0,C 180,E1 -3033.902,E2 -3033.902} C_VEL
LIN {X 0,Y 559.12,Z 233.836,A -85,B 0,C 180,E1 -3037.066,E2 -3037.066} C_VEL
LIN {X 0,Y 559.179,Z 233.834,A -85,B 0,C 180,E1 -3039.395,E2 -3039.395} C_VEL
LIN {X 0,Y 559.145,Z 233.834,A -85,B 0,C 180,E1 -3041.686,E2 -3041.686} C_VEL
LIN {X 0,Y 559.162,Z 233.832,A -85,B 0,C 180,E1 -3043.948,E2 -3043.948} C_VEL
LIN {X 0,Y 559.16,Z 233.837,A -85,B 0,C 180,E1 -3046.184,E2 -3046.184} C_VEL
LIN {X 0,Y 559.182,Z 233.829,A -85,B 0,C 180,E1 -3049.133,E2 -3049.133} C_VEL
LIN {X 0,Y 559.179,Z 233.829,A -85,B 0,C 180,E1 -3052.053,E2 -3052.053} C_VEL
LIN {X 0,Y 559.255,Z 233.826,A -85,B 0,C 180,E1 -3054.953,E2 -3054.953} C_VEL
LIN {X 0,Y 559.254,Z 233.822,A -85,B 0,C 180,E1 -3057.839,E2 -3057.839} C_VEL
LIN {X 0,Y 559.262,Z 233.819,A -85,B 0,C 180,E1 -3060.72,E2 -3060.72} C_VEL
LIN {X 0,Y 559.219,Z 233.825,A -85,B 0,C 180,E1 -3062.882,E2 -3062.882} C_VEL
LIN {X 0,Y 559.214,Z 233.824,A -85,B 0,C 180,E1 -3065.77,E2 -3065.77} C_VEL
LIN {X 0,Y 559.174,Z 233.835,A -85,B 0,C 180,E1 -3068.675,E2 -3068.675} C_VEL
LIN {X 0,Y 559.209,Z 233.828,A -85,B 0,C 180,E1 -3071.6,E2 -3071.6} C_VEL
LIN {X 0,Y 559.183,Z 233.829,A -85,B 0,C 180,E1 -3074.588,E2 -3074.588} C_VEL
LIN {X 0,Y 559.132,Z 233.836,A -85,B 0,C 180,E1 -3077.558,E2 -3077.558} C_VEL
LIN {X 0,Y 559.166,Z 233.83,A -85,B 0,C 180,E1 -3079.838,E2 -3079.838} C_VEL
LIN {X 0,Y 559.142,Z 233.838,A -85,B 0,C 180,E1 -3082.153,E2 -3082.153} C_VEL
LIN {X 0,Y 559.179,Z 233.831,A -85,B 0,C 180,E1 -3085.298,E2 -3085.298} C_VEL
LIN {X 0,Y 559.149,Z 233.836,A -85,B 0,C 180,E1 -3087.714,E2 -3087.714} C_VEL
LIN {X 0,Y 559.125,Z 233.836,A -85,B 0,C 180,E1 -3090.598,E2 -3090.598} C_VEL
LIN {X 0,Y 558.469,Z 233.921,A -85,B 0,C 180,E1 -3091.199,E2 -3091.199} C_VEL
LIN {X 0,Y 555.611,Z 234.276,A -85,B 0,C 180,E1 -3092.176,E2 -3092.176} C_VEL
LIN {X 0,Y 553.194,Z 234.576,A -85,B 0,C 180,E1 -3092.961,E2 -3092.961} C_VEL
LIN {X 0,Y 552.166,Z 234.703,A -85,B 0,C 180,E1 -3093.568,E2 -3093.568} C_VEL
LIN {X 0,Y 552.087,Z 234.713,A -85,B 0,C 180,E1 -3093.774,E2 -3093.774} C_VEL
LIN {X 0,Y 552.1,Z 234.71,A -85,B 0,C 180,E1 -3096.748,E2 -3096.748} C_VEL
LIN {X 0,Y 552.131,Z 234.713,A -85,B 0,C 180,E1 -3099.527,E2 -3099.527} C_VEL
LIN {X 0,Y 552.111,Z 234.712,A -85,B 0,C 180,E1 -3102.428,E2 -3102.428} C_VEL
LIN {X 0,Y 552.068,Z 234.715,A -85,B 0,C 180,E1 -3105.559,E2 -3105.559} C_VEL
LIN {X 0,Y 552.07,Z 234.715,A -85,B 0,C 180,E1 -3108.549,E2 -3108.549} C_VEL
LIN {X 0,Y 552.119,Z 234.715,A -85,B 0,C 180,E1 -3111.411,E2 -3111.411} C_VEL
LIN {X 0,Y 552.059,Z 234.717,A -85,B 0,C 180,E1 -3114.154,E2 -3114.154} C_VEL
LIN {X 0,Y 552.025,Z 234.724,A -85,B 0,C 180,E1 -3114.568,E2 -3114.568} C_VEL
LIN {X 0,Y 552.033,Z 238.07,A -85,B 0,C 180,E1 -3116.809,E2 -3116.809} C_VEL
LIN {X 0,Y 551.957,Z 242.174,A -85,B 0,C 180,E1 -3119.382,E2 -3119.382} C_VEL
LIN {X 0,Y 551.951,Z 246.247,A -85,B 0,C 180,E1 -3121.893,E2 -3121.893} C_VEL
LIN {X 0,Y 551.905,Z 251.665,A -85,B 0,C 180,E1 -3125.151,E2 -3125.151} C_VEL
LIN {X 0,Y 551.87,Z 257.065,A -85,B 0,C 180,E1 -3128.327,E2 -3128.327} C_VEL
LIN {X 0,Y 551.76,Z 262.487,A -85,B 0,C 180,E1 -3131.432,E2 -3131.432} C_VEL
LIN {X 0,Y 551.74,Z 266.511,A -85,B 0,C 180,E1 -3133.726,E2 -3133.726} C_VEL
LIN {X 0,Y 551.733,Z 270.546,A -85,B 0,C 180,E1 -3135.994,E2 -3135.994} C_VEL
LIN {X 0,Y 551.725,Z 272.533,A -85,B 0,C 180,E1 -3137.073,E2 -3137.073} C_VEL
LIN {X 0,Y 553.048,Z 281.324,A -85,B 0,C 180,E1 -3137.314,E2 -3137.314} C_VEL
LIN {X 0,Y 552.867,Z 294.313,A -85,B 0,C 180,E1 -3137.725,E2 -3137.725} C_VEL
LIN {X 0,Y 552.737,Z 306.317,A -85,B 0,C 180,E1 -3138.262,E2 -3138.262} C_VEL
LIN {X 0,Y 552.547,Z 317.751,A -85,B 0,C 180,E1 -3138.926,E2 -3138.926} C_VEL
LIN {X 0,Y 552.361,Z 328.86,A -85,B 0,C 180,E1 -3139.739,E2 -3139.739} C_VEL
LIN {X 0,Y 552.175,Z 338.9,A -85,B 0,C 180,E1 -3140.661,E2 -3140.661} C_VEL
LIN {X 0,Y 552.007,Z 348.6,A -85,B 0,C 180,E1 -3141.765,E2 -3141.765} C_VEL
LIN {X 0,Y 551.895,Z 356.461,A -85,B 0,C 180,E1 -3142.886,E2 -3142.886} C_VEL
LIN {X 0,Y 551.868,Z 363.457,A -85,B 0,C 180,E1 -3144.153,E2 -3144.153} C_VEL
LIN {X 0,Y 551.725,Z 368.197,A -85,B 0,C 180,E1 -3145.251,E2 -3145.251} C_VEL
LIN {X 0,Y 551.75,Z 371.83,A -85,B 0,C 180,E1 -3146.349,E2 -3146.349} C_VEL
LIN {X 0,Y 551.723,Z 373.706,A -85,B 0,C 180,E1 -3147.079,E2 -3147.079} C_VEL
LIN {X 0,Y 551.656,Z 375.128,A -85,B 0,C 180,E1 -3147.81,E2 -3147.81} C_VEL
LIN {X 0,Y 551.642,Z 376.757,A -85,B 0,C 180,E1 -3149.27,E2 -3149.27} C_VEL
LIN {X 0,Y 551.641,Z 376.996,A -85,B 0,C 180,E1 -3150,E2 -3150} C_VEL
LIN {X 0,Y 551.641,Z 376.815,A -85,B 0,C 180,E1 -3150.73,E2 -3150.73} C_VEL
LIN {X 0,Y 551.655,Z 375.264,A -85,B 0,C 180,E1 -3152.19,E2 -3152.19} C_VEL
LIN {X 0,Y 551.724,Z 373.903,A -85,B 0,C 180,E1 -3152.921,E2 -3152.921} C_VEL
LIN {X 0,Y 551.764,Z 371.025,A -85,B 0,C 180,E1 -3154.017,E2 -3154.017} C_VEL
LIN {X 0,Y 551.723,Z 367.124,A -85,B 0,C 180,E1 -3155.116,E2 -3155.116} C_VEL
LIN {X 0,Y 551.811,Z 361.393,A -85,B 0,C 180,E1 -3156.349,E2 -3156.349} C_VEL
LIN {X 0,Y 551.925,Z 354.536,A -85,B 0,C 180,E1 -3157.5,E2 -3157.5} C_VEL
LIN {X 0,Y 552.063,Z 346.354,A -85,B 0,C 180,E1 -3158.603,E2 -3158.603} C_VEL
LIN {X 0,Y 552.197,Z 337.985,A -85,B 0,C 180,E1 -3159.524,E2 -3159.524} C_VEL
LIN {X 0,Y 552.389,Z 327.661,A -85,B 0,C 180,E1 -3160.446,E2 -3160.446} C_VEL
LIN {X 0,Y 552.547,Z 316.979,A -85,B 0,C 180,E1 -3161.214,E2 -3161.214} C_VEL
LIN {X 0,Y 552.745,Z 306.258,A -85,B 0,C 180,E1 -3161.831,E2 -3161.831} C_VEL
LIN {X 0,Y 552.901,Z 293.726,A -85,B 0,C 180,E1 -3162.386,E2 -3162.386} C_VEL
LIN {X 0,Y 553.028,Z 280.281,A -85,B 0,C 180,E1 -3162.803,E2 -3162.803} C_VEL
LIN {X 0,Y 551.699,Z 272.526,A -85,B 0,C 180,E1 -3163.022,E2 -3163.022} C_VEL
LIN {X 0,Y 551.745,Z 268.003,A -85,B 0,C 180,E1 -3165.515,E2 -3165.515} C_VEL
LIN {X 0,Y 551.767,Z 263.994,A -85,B 0,C 180,E1 -3167.8,E2 -3167.8} C_VEL
LIN {X 0,Y 551.797,Z 259.939,A -85,B 0,C 180,E1 -3170.114,E2 -3170.114} C_VEL
LIN {X 0,Y 551.842,Z 255.87,A -85,B 0,C 180,E1 -3172.462,E2 -3172.462} C_VEL
LIN {X 0,Y 551.905,Z 251.068,A -85,B 0,C 180,E1 -3175.295,E2 -3175.295} C_VEL
LIN {X 0,Y 551.951,Z 246.394,A -85,B 0,C 180,E1 -3178.107,E2 -3178.107} C_VEL
LIN {X 0,Y 551.954,Z 242.323,A -85,B 0,C 180,E1 -3180.619,E2 -3180.619} C_VEL
LIN {X 0,Y 552.014,Z 238.215,A -85,B 0,C 180,E1 -3183.193,E2 -3183.193} C_VEL
LIN {X 0,Y 552.032,Z 234.724,A -85,B 0,C 180,E1 -3185.433,E2 -3185.433} C_VEL
LIN {X 0,Y 552.1,Z 234.71,A -85,B 0,C 180,E1 -3187.886,E2 -3187.886} C_VEL
LIN {X 0,Y 552.11,Z 234.715,A -85,B 0,C 180,E1 -3190.481,E2 -3190.481} C_VEL
LIN {X 0,Y 552.061,Z 234.718,A -85,B 0,C 180,E1 -3193.478,E2 -3193.478} C_VEL
LIN {X 0,Y 552.075,Z 234.715,A -85,B 0,C 180,E1 -3196.573,E2 -3196.573} C_VEL
LIN {X 0,Y 552.111,Z 234.71,A -85,B 0,C 180,E1 -3199.519,E2 -3199.519} C_VEL
LIN {X 0,Y 552.095,Z 234.718,A -85,B 0,C 180,E1 -3202.336,E2 -3202.336} C_VEL
LIN {X 0,Y 552.084,Z 234.712,A -85,B 0,C 180,E1 -3205.051,E2 -3205.051} C_VEL
LIN {X 0,Y 552.115,Z 234.714,A -85,B 0,C 180,E1 -3207.681,E2 -3207.681} C_VEL
LIN {X 0,Y 552.082,Z 234.713,A -85,B 0,C 180,E1 -3210.233,E2 -3210.233} C_VEL
LIN {X 0,Y 552.141,Z 234.709,A -85,B 0,C 180,E1 -3213,E2 -3213} C_VEL
LIN {X 0,Y 552.117,Z 234.709,A -85,B 0,C 180,E1 -3215.161,E2 -3215.161} C_VEL
LIN {X 0,Y 552.13,Z 234.707,A -85,B 0,C 180,E1 -3218.337,E2 -3218.337} C_VEL
LIN {X 0,Y 552.153,Z 234.704,A -85,B 0,C 180,E1 -3220.674,E2 -3220.674} C_VEL
LIN {X 0,Y 552.088,Z 234.712,A -85,B 0,C 180,E1 -3223.736,E2 -3223.736} C_VEL
LIN {X 0,Y 552.125,Z 234.711,A -85,B 0,C 180,E1 -3226.004,E2 -3226.004} C_VEL
LIN {X 0,Y 552.165,Z 234.703,A -85,B 0,C 180,E1 -3228.993,E2 -3228.993} C_VEL
LIN {X 0,Y 552.15,Z 234.706,A -85,B 0,C 180,E1 -3231.951,E2 -3231.951} C_VEL
LIN {X 0,Y 552.217,Z 234.702,A -85,B 0,C 180,E1 -3234.889,E2 -3234.889} C_VEL
LIN {X 0,Y 552.21,Z 234.698,A -85,B 0,C 180,E1 -3237.812,E2 -3237.812} C_VEL
LIN {X 0,Y 552.242,Z 234.694,A -85,B 0,C 180,E1 -3240.729,E2 -3240.729} C_VEL
LIN {X 0,Y 552.208,Z 234.699,A -85,B 0,C 180,E1 -3242.918,E2 -3242.918} C_VEL
LIN {X 0,Y 552.197,Z 234.699,A -85,B 0,C 180,E1 -3245.844,E2 -3245.844} C_VEL
LIN {X 0,Y 552.133,Z 234.71,A -85,B 0,C 180,E1 -3248.786,E2 -3248.786} C_VEL
LIN {X 0,Y 552.113,Z 234.712,A -85,B 0,C 180,E1 -3251.752,E2 -3251.752} C_VEL
LIN {X 0,Y 552.132,Z 234.707,A -85,B 0,C 180,E1 -3254.749,E2 -3254.749} C_VEL
LIN {X 0,Y 552.113,Z 234.71,A -85,B 0,C 180,E1 -3257.788,E2 -3257.788} C_VEL
LIN {X 0,Y 552.131,Z 234.708,A -85,B 0,C 180,E1 -3260.101,E2 -3260.101} C_VEL
LIN {X 0,Y 552.093,Z 234.716,A -85,B 0,C 180,E1 -3262.451,E2 -3262.451} C_VEL
LIN {X 0,Y 552.084,Z 234.714,A -85,B 0,C 180,E1 -3265.334,E2 -3265.334} C_VEL
LIN {X 0,Y 552.079,Z 234.714,A -85,B 0,C 180,E1 -3268.1,E2 -3268.1} C_VEL
LIN {X 0,Y 552.099,Z 234.715,A -85,B 0,C 180,E1 -3270.61,E2 -3270.61} C_VEL
LIN {X 0,Y 552.119,Z 234.709,A -85,B 0,C 180,E1 -3273.186,E2 -3273.186} C_VEL
LIN {X 0,Y 552.077,Z 234.719,A -85,B 0,C 180,E1 -3275.844,E2 -3275.844} C_VEL
LIN {X 0,Y 552.111,Z 234.708,A -85,B 0,C 180,E1 -3278.59,E2 -3278.59} C_VEL
LIN {X 0,Y 552.077,Z 234.717,A -85,B 0,C 180,E1 -3281.45,E2 -3281.45} C_VEL
LIN {X 0,Y 552.094,Z 234.717,A -85,B 0,C 180,E1 -3284.438,E2 -3284.438} C_VEL
LIN {X 0,Y 552.133,Z 234.709,A -85,B 0,C 180,E1 -3287.585,E2 -3287.585} C_VEL
LIN {X 0,Y 552.13,Z 234.709,A -85,B 0,C 180,E1 -3290.473,E2 -3290.473} C_VEL
LIN {X 0,Y 552.15,Z 234.848,A -85,B 0,C 180,E1 -3293.311,E2 -3293.311} C_VEL
LIN {X 0,Y 552.522,Z 239.082,A -85,B 0,C 180,E1 -3295.082,E2 -3295.082} C_VEL
LIN {X 0,Y 552.439,Z 245.69,A -85,B 0,C 180,E1 -3297.702,E2 -3297.702} C_VEL
LIN {X 0,Y 552.294,Z 253.542,A -85,B 0,C 180,E1 -3300.665,E2 -3300.665} C_VEL
LIN {X 0,Y 552.16,Z 261.41,A -85,B 0,C 180,E1 -3303.545,E2 -3303.545} C_VEL
LIN {X 0,Y 552.114,Z 269.503,A -85,B 0,C 180,E1 -3306.421,E2 -3306.421} C_VEL
LIN {X 0,Y 552.019,Z 277.192,A -85,B 0,C 180,E1 -3309.116,E2 -3309.116} C_VEL
LIN {X 0,Y 551.945,Z 285.103,A -85,B 0,C 180,E1 -3311.822,E2 -3311.822} C_VEL
LIN {X 0,Y 551.903,Z 293.048,A -85,B 0,C 180,E1 -3314.489,E2 -3314.489} C_VEL
LIN {X 0,Y 551.838,Z 300.491,A -85,B 0,C 180,E1 -3317.005,E2 -3317.005} C_VEL
LIN {X 0,Y 553.087,Z 309.431,A -85,B 0,C 180,E1 -3317.222,E2 -3317.222} C_VEL
LIN {X 0,Y 552.935,Z 322.471,A -85,B 0,C 180,E1 -3317.614,E2 -3317.614} C_VEL
LIN {X 0,Y 552.74,Z 333.488,A -85,B 0,C 180,E1 -3318.076,E2 -3318.076} C_VEL
LIN {X 0,Y 552.542,Z 345.375,A -85,B 0,C 180,E1 -3318.726,E2 -3318.726} C_VEL
LIN {X 0,Y 552.425,Z 357.092,A -85,B 0,C 180,E1 -3319.555,E2 -3319.555} C_VEL
LIN {X 0,Y 552.201,Z 367.538,A -85,B 0,C 180,E1 -3320.476,E2 -3320.476} C_VEL
LIN {X 0,Y 552.082,Z 375.991,A -85,B 0,C 180,E1 -3321.397,E2 -3321.397} C_VEL
LIN {X 0,Y 551.926,Z 384.235,A -85,B 0,C 180,E1 -3322.5,E2 -3322.5} C_VEL
LIN {X 0,Y 551.821,Z 391.207,A -85,B 0,C 180,E1 -3323.662,E2 -3323.662} C_VEL
LIN {X 0,Y 551.724,Z 396.949,A -85,B 0,C 180,E1 -3324.884,E2 -3324.884} C_VEL
LIN {X 0,Y 551.764,Z 400.894,A -85,B 0,C 180,E1 -3325.983,E2 -3325.983} C_VEL
LIN {X 0,Y 551.723,Z 403.807,A -85,B 0,C 180,E1 -3327.079,E2 -3327.079} C_VEL
LIN {X 0,Y 551.645,Z 406.183,A -85,B 0,C 180,E1 -3328.54,E2 -3328.54} C_VEL
LIN {X 0,Y 551.64,Z 407,A -85,B 0,C 180,E1 -3330,E2 -3330} C_VEL
LIN {X 0,Y 551.645,Z 406.185,A -85,B 0,C 180,E1 -3331.46,E2 -3331.46} C_VEL
LIN {X 0,Y 551.723,Z 403.81,A -85,B 0,C 180,E1 -3332.921,E2 -3332.921} C_VEL
LIN {X 0,Y 551.764,Z 400.896,A -85,B 0,C 180,E1 -3334.017,E2 -3334.017} C_VEL
LIN {X 0,Y 551.723,Z 396.949,A -85,B 0,C 180,E1 -3335.116,E2 -3335.116} C_VEL
LIN {X 0,Y 551.815,Z 391.123,A -85,B 0,C 180,E1 -3336.353,E2 -3336.353} C_VEL
LIN {X 0,Y 551.926,Z 384.236,A -85,B 0,C 180,E1 -3337.5,E2 -3337.5} C_VEL
LIN {X 0,Y 552.082,Z 375.992,A -85,B 0,C 180,E1 -3338.602,E2 -3338.602} C_VEL
LIN {X 0,Y 552.2,Z 367.54,A -85,B 0,C 180,E1 -3339.524,E2 -3339.524} C_VEL
LIN {X 0,Y 552.425,Z 357.093,A -85,B 0,C 180,E1 -3340.445,E2 -3340.445} C_VEL
LIN {X 0,Y 552.553,Z 346.41,A -85,B 0,C 180,E1 -3341.206,E2 -3341.206} C_VEL
LIN {X 0,Y 552.702,Z 335.406,A -85,B 0,C 180,E1 -3341.832,E2 -3341.832} C_VEL
LIN {X 0,Y 552.865,Z 323.764,A -85,B 0,C 180,E1 -3342.34,E2 -3342.34} C_VEL
LIN {X 0,Y 553.075,Z 310.345,A -85,B 0,C 180,E1 -3342.755,E2 -3342.755} C_VEL
LIN {X 0,Y 552.525,Z 304.673,A -85,B 0,C 180,E1 -3342.896,E2 -3342.896} C_VEL
LIN {X 0,Y 551.838,Z 300.492,A -85,B 0,C 180,E1 -3342.995,E2 -3342.995} C_VEL
LIN {X 0,Y 551.903,Z 291.918,A -85,B 0,C 180,E1 -3345.89,E2 -3345.89} C_VEL
LIN {X 0,Y 551.983,Z 282.828,A -85,B 0,C 180,E1 -3348.946,E2 -3348.946} C_VEL
LIN {X 0,Y 552.076,Z 274.925,A -85,B 0,C 180,E1 -3351.674,E2 -3351.674} C_VEL
LIN {X 0,Y 552.143,Z 267.081,A -85,B 0,C 180,E1 -3354.436,E2 -3354.436} C_VEL
LIN {X 0,Y 552.18,Z 259.164,A -85,B 0,C 180,E1 -3357.271,E2 -3357.271} C_VEL
LIN {X 0,Y 552.301,Z 251.534,A -85,B 0,C 180,E1 -3360.083,E2 -3360.083} C_VEL
LIN {X 0,Y 552.455,Z 244.13,A -85,B 0,C 180,E1 -3362.9,E2 -3362.9} C_VEL
LIN {X 0,Y 552.513,Z 237.644,A -85,B 0,C 180,E1 -3365.503,E2 -3365.503} C_VEL
LIN {X 0,Y 552.117,Z 234.716,A -85,B 0,C 180,E1 -3366.746,E2 -3366.746} C_VEL
LIN {X 0,Y 552.129,Z 234.709,A -85,B 0,C 180,E1 -3369.527,E2 -3369.527} C_VEL
LIN {X 0,Y 552.133,Z 234.709,A -85,B 0,C 180,E1 -3372.425,E2 -3372.425} C_VEL
LIN {X 0,Y 552.095,Z 234.717,A -85,B 0,C 180,E1 -3375.562,E2 -3375.562} C_VEL
LIN {X 0,Y 552.076,Z 234.716,A -85,B 0,C 180,E1 -3378.55,E2 -3378.55} C_VEL
LIN {X 0,Y 552.11,Z 234.709,A -85,B 0,C 180,E1 -3381.41,E2 -3381.41} C_VEL
LIN {X 0,Y 552.076,Z 234.719,A -85,B 0,C 180,E1 -3384.155,E2 -3384.155} C_VEL
LIN {X 0,Y 552.124,Z 234.709,A -85,B 0,C 180,E1 -3386.815,E2 -3386.815} C_VEL
LIN {X 0,Y 552.105,Z 234.714,A -85,B 0,C 180,E1 -3389.391,E2 -3389.391} C_VEL
LIN {X 0,Y 552.079,Z 234.714,A -85,B 0,C 180,E1 -3391.9,E2 -3391.9} C_VEL
LIN {X 0,Y 552.083,Z 234.714,A -85,B 0,C 180,E1 -3394.666,E2 -3394.666} C_VEL
LIN {X 0,Y 552.092,Z 234.716,A -85,B 0,C 180,E1 -3397.549,E2 -3397.549} C_VEL
LIN {X 0,Y 552.147,Z 234.705,A -85,B 0,C 180,E1 -3400.375,E2 -3400.375} C_VEL
LIN {X 0,Y 552.157,Z 234.709,A -85,B 0,C 180,E1 -3402.977,E2 -3402.977} C_VEL
LIN {X 0,Y 552.128,Z 234.711,A -85,B 0,C 180,E1 -3406.004,E2 -3406.004} C_VEL
LIN {X 0,Y 552.154,Z 234.704,A -85,B 0,C 180,E1 -3408.993,E2 -3408.993} C_VEL
LIN {X 0,Y 552.137,Z 234.707,A -85,B 0,C 180,E1 -3411.951,E2 -3411.951} C_VEL
LIN {X 0,Y 552.229,Z 234.701,A -85,B 0,C 180,E1 -3414.889,E2 -3414.889} C_VEL
LIN {X 0,Y 552.226,Z 234.697,A -85,B 0,C 180,E1 -3417.812,E2 -3417.812} C_VEL
LIN {X 0,Y 552.234,Z 234.694,A -85,B 0,C 180,E1 -3420.729,E2 -3420.729} C_VEL
LIN {X 0,Y 552.187,Z 234.701,A -85,B 0,C 180,E1 -3422.918,E2 -3422.918} C_VEL
LIN {X 0,Y 552.183,Z 234.7,A -85,B 0,C 180,E1 -3425.844,E2 -3425.844} C_VEL
LIN {X 0,Y 552.15,Z 234.709,A -85,B 0,C 180,E1 -3428.786,E2 -3428.786} C_VEL
LIN {X 0,Y 552.166,Z 234.707,A -85,B 0,C 180,E1 -3431.751,E2 -3431.751} C_VEL
LIN {X 0,Y 552.131,Z 234.708,A -85,B 0,C 180,E1 -3434.749,E2 -3434.749} C_VEL
LIN {X 0,Y 552.09,Z 234.712,A -85,B 0,C 180,E1 -3437.789,E2 -3437.789} C_VEL
LIN {X 0,Y 552.127,Z 234.708,A -85,B 0,C 180,E1 -3440.101,E2 -3440.101} C_VEL
LIN {X 0,Y 552.094,Z 234.716,A -85,B 0,C 180,E1 -3442.451,E2 -3442.451} C_VEL
LIN {X 0,Y 552.159,Z 234.706,A -85,B 0,C 180,E1 -3445.351,E2 -3445.351} C_VEL
LIN {X 0,Y 552.094,Z 234.712,A -85,B 0,C 180,E1 -3448.099,E2 -3448.099} C_VEL
LIN {X 0,Y 552.09,Z 234.716,A -85,B 0,C 180,E1 -3450.61,E2 -3450.61} C_VEL
LIN {X 0,Y 552.106,Z 234.71,A -85,B 0,C 180,E1 -3453.187,E2 -3453.187} C_VEL
LIN {X 0,Y 552.087,Z 234.713,A -85,B 0,C 180,E1 -3453.774,E2 -3453.774} C_VEL
LIN {X 0,Y 551.446,Z 234.797,A -85,B 0,C 180,E1 -3454.382,E2 -3454.382} C_VEL
LIN {X 0,Y 548.632,Z 235.145,A -85,B 0,C 180,E1 -3455.37,E2 -3455.37} C_VEL
LIN {X 0,Y 546.224,Z 235.447,A -85,B 0,C 180,E1 -3456.166,E2 -3456.166} C_VEL
LIN {X 0,Y 545.161,Z 235.575,A -85,B 0,C 180,E1 -3456.78,E2 -3456.78} C_VEL
LIN {X 0,Y 545.06,Z 235.587,A -85,B 0,C 180,E1 -3456.988,E2 -3456.988} C_VEL
LIN {X 0,Y 545.067,Z 235.587,A -85,B 0,C 180,E1 -3460.143,E2 -3460.143} C_VEL
LIN {X 0,Y 545.041,Z 235.595,A -85,B 0,C 180,E1 -3462.694,E2 -3462.694} C_VEL
LIN {X 0,Y 545.018,Z 235.594,A -85,B 0,C 180,E1 -3465.172,E2 -3465.172} C_VEL
LIN {X 0,Y 545.036,Z 235.597,A -85,B 0,C 180,E1 -3467.893,E2 -3467.893} C_VEL
LIN {X 0,Y 545.081,Z 235.585,A -85,B 0,C 180,E1 -3470.818,E2 -3470.818} C_VEL
LIN {X 0,Y 545.033,Z 235.593,A -85,B 0,C 180,E1 -3473.619,E2 -3473.619} C_VEL
LIN {X 0,Y 544.991,Z 235.6,A -85,B 0,C 180,E1 -3474.528,E2 -3474.528} C_VEL
LIN {X 0,Y 545.013,Z 238.135,A -85,B 0,C 180,E1 -3476.324,E2 -3476.324} C_VEL
LIN {X 0,Y 544.925,Z 242.258,A -85,B 0,C 180,E1 -3478.943,E2 -3478.943} C_VEL
LIN {X 0,Y 544.941,Z 246.344,A -85,B 0,C 180,E1 -3481.498,E2 -3481.498} C_VEL
LIN {X 0,Y 544.859,Z 251.773,A -85,B 0,C 180,E1 -3484.808,E2 -3484.808} C_VEL
LIN {X 0,Y 544.799,Z 257.19,A -85,B 0,C 180,E1 -3488.031,E2 -3488.031} C_VEL
LIN {X 0,Y 544.697,Z 262.611,A -85,B 0,C 180,E1 -3491.182,E2 -3491.182} C_VEL
LIN {X 0,Y 544.698,Z 266.684,A -85,B 0,C 180,E1 -3493.51,E2 -3493.51} C_VEL
LIN {X 0,Y 544.668,Z 270.696,A -85,B 0,C 180,E1 -3495.809,E2 -3495.809} C_VEL
LIN {X 0,Y 544.618,Z 272.628,A -85,B 0,C 180,E1 -3496.901,E2 -3496.901} C_VEL
LIN {X 0,Y 546.117,Z 282.31,A -85,B 0,C 180,E1 -3497.174,E2 -3497.174} C_VEL
LIN {X 0,Y 545.93,Z 295.055,A -85,B 0,C 180,E1 -3497.595,E2 -3497.595} C_VEL
LIN {X 0,Y 545.783,Z 306.871,A -85,B 0,C 180,E1 -3498.139,E2 -3498.139} C_VEL
LIN {X 0,Y 545.549,Z 318.916,A -85,B 0,C 180,E1 -3498.858,E2 -3498.858} C_VEL
LIN {X 0,Y 545.311,Z 329.953,A -85,B 0,C 180,E1 -3499.699,E2 -3499.699} C_VEL
LIN {X 0,Y 545.122,Z 340.686,A -85,B 0,C 180,E1 -3500.726,E2 -3500.726} C_VEL
LIN {X 0,Y 544.975,Z 348.604,A -85,B 0,C 180,E1 -3501.658,E2 -3501.658} C_VEL
LIN {X 0,Y 544.829,Z 356.353,A -85,B 0,C 180,E1 -3502.775,E2 -3502.775} C_VEL
LIN {X 0,Y 544.778,Z 363.46,A -85,B 0,C 180,E1 -3504.076,E2 -3504.076} C_VEL
LIN {X 0,Y 544.629,Z 368.199,A -85,B 0,C 180,E1 -3505.189,E2 -3505.189} C_VEL
LIN {X 0,Y 544.669,Z 371.831,A -85,B 0,C 180,E1 -3506.301,E2 -3506.301} C_VEL
LIN {X 0,Y 544.65,Z 373.708,A -85,B 0,C 180,E1 -3507.041,E2 -3507.041} C_VEL
LIN {X 0,Y 544.57,Z 375.128,A -85,B 0,C 180,E1 -3507.781,E2 -3507.781} C_VEL
LIN {X 0,Y 544.542,Z 376.757,A -85,B 0,C 180,E1 -3509.261,E2 -3509.261} C_VEL
LIN {X 0,Y 544.541,Z 376.996,A -85,B 0,C 180,E1 -3510,E2 -3510} C_VEL
LIN {X 0,Y 544.542,Z 376.814,A -85,B 0,C 180,E1 -3510.74,E2 -3510.74} C_VEL
LIN {X 0,Y 544.57,Z 375.262,A -85,B 0,C 180,E1 -3512.219,E2 -3512.219} C_VEL
LIN {X 0,Y 544.651,Z 373.901,A -85,B 0,C 180,E1 -3512.959,E2 -3512.959} C_VEL
LIN {X 0,Y 544.684,Z 371.023,A -85,B 0,C 180,E1 -3514.07,E2 -3514.07} C_VEL
LIN {X 0,Y 544.653,Z 367.122,A -85,B 0,C 180,E1 -3515.182,E2 -3515.182} C_VEL
LIN {X 0,Y 544.725,Z 361.897,A -85,B 0,C 180,E1 -3516.335,E2 -3516.335} C_VEL
LIN {X 0,Y 544.859,Z 354.531,A -85,B 0,C 180,E1 -3517.598,E2 -3517.598} C_VEL
LIN {X 0,Y 544.999,Z 346.349,A -85,B 0,C 180,E1 -3518.715,E2 -3518.715} C_VEL
LIN {X 0,Y 545.16,Z 337.978,A -85,B 0,C 180,E1 -3519.648,E2 -3519.648} C_VEL
LIN {X 0,Y 545.367,Z 327.652,A -85,B 0,C 180,E1 -3520.582,E2 -3520.582} C_VEL
LIN {X 0,Y 545.596,Z 316.265,A -85,B 0,C 180,E1 -3521.406,E2 -3521.406} C_VEL
LIN {X 0,Y 545.817,Z 304.444,A -85,B 0,C 180,E1 -3522.078,E2 -3522.078} C_VEL
LIN {X 0,Y 545.994,Z 292.443,A -85,B 0,C 180,E1 -3522.593,E2 -3522.593} C_VEL
LIN {X 0,Y 545.987,Z 280.312,A -85,B 0,C 180,E1 -3522.971,E2 -3522.971} C_VEL
LIN {X 0,Y 544.623,Z 272.614,A -85,B 0,C 180,E1 -3523.194,E2 -3523.194} C_VEL
LIN {X 0,Y 544.68,Z 269.506,A -85,B 0,C 180,E1 -3524.955,E2 -3524.955} C_VEL
LIN {X 0,Y 544.721,Z 265.424,A -85,B 0,C 180,E1 -3527.302,E2 -3527.302} C_VEL
LIN {X 0,Y 544.742,Z 260.06,A -85,B 0,C 180,E1 -3530.386,E2 -3530.386} C_VEL
LIN {X 0,Y 544.792,Z 255.992,A -85,B 0,C 180,E1 -3532.769,E2 -3532.769} C_VEL
LIN {X 0,Y 544.835,Z 251.496,A -85,B 0,C 180,E1 -3535.451,E2 -3535.451} C_VEL
LIN {X 0,Y 544.942,Z 246.491,A -85,B 0,C 180,E1 -3538.502,E2 -3538.502} C_VEL
LIN {X 0,Y 544.936,Z 241.455,A -85,B 0,C 180,E1 -3541.657,E2 -3541.657} C_VEL
LIN {X 0,Y 544.999,Z 236.88,A -85,B 0,C 180,E1 -3544.569,E2 -3544.569} C_VEL
LIN {X 0,Y 544.997,Z 235.6,A -85,B 0,C 180,E1 -3545.472,E2 -3545.472} C_VEL
LIN {X 0,Y 545.053,Z 235.589,A -85,B 0,C 180,E1 -3548.136,E2 -3548.136} C_VEL
LIN {X 0,Y 545.082,Z 235.591,A -85,B 0,C 180,E1 -3550.472,E2 -3550.472} C_VEL
LIN {X 0,Y 545.019,Z 235.593,A -85,B 0,C 180,E1 -3553.113,E2 -3553.113} C_VEL
LIN {X 0,Y 545.047,Z 235.59,A -85,B 0,C 180,E1 -3556.227,E2 -3556.227} C_VEL
LIN {X 0,Y 545.084,Z 235.59,A -85,B 0,C 180,E1 -3558.885,E2 -3558.885} C_VEL
LIN {X 0,Y 545.054,Z 235.589,A -85,B 0,C 180,E1 -3561.763,E2 -3561.763} C_VEL
LIN {X 0,Y 545.039,Z 235.591,A -85,B 0,C 180,E1 -3564.532,E2 -3564.532} C_VEL
LIN {X 0,Y 545.067,Z 235.59,A -85,B 0,C 180,E1 -3567.211,E2 -3567.211} C_VEL
LIN {X 0,Y 545.065,Z 235.588,A -85,B 0,C 180,E1 -3569.81,E2 -3569.81} C_VEL
LIN {X 0,Y 545.088,Z 235.589,A -85,B 0,C 180,E1 -3572.829,E2 -3572.829} C_VEL
LIN {X 0,Y 545.053,Z 235.59,A -85,B 0,C 180,E1 -3575.631,E2 -3575.631} C_VEL
LIN {X 0,Y 545.068,Z 235.586,A -85,B 0,C 180,E1 -3578.837,E2 -3578.837} C_VEL
LIN {X 0,Y 545.052,Z 235.594,A -85,B 0,C 180,E1 -3581.195,E2 -3581.195} C_VEL
LIN {X 0,Y 545.039,Z 235.591,A -85,B 0,C 180,E1 -3583.52,E2 -3583.52} C_VEL
LIN {X 0,Y 545.088,Z 235.586,A -85,B 0,C 180,E1 -3585.82,E2 -3585.82} C_VEL
LIN {X 0,Y 545.121,Z 235.581,A -85,B 0,C 180,E1 -3588.849,E2 -3588.849} C_VEL
LIN {X 0,Y 545.099,Z 235.585,A -85,B 0,C 180,E1 -3591.847,E2 -3591.847} C_VEL
LIN {X 0,Y 545.193,Z 235.576,A -85,B 0,C 180,E1 -3594.823,E2 -3594.823} C_VEL
LIN {X 0,Y 545.183,Z 235.573,A -85,B 0,C 180,E1 -3597.784,E2 -3597.784} C_VEL
LIN {X 0,Y 545.213,Z 235.569,A -85,B 0,C 180,E1 -3600.739,E2 -3600.739} C_VEL
LIN {X 0,Y 545.174,Z 235.575,A -85,B 0,C 180,E1 -3602.956,E2 -3602.956} C_VEL
LIN {X 0,Y 545.169,Z 235.574,A -85,B 0,C 180,E1 -3605.92,E2 -3605.92} C_VEL
LIN {X 0,Y 545.093,Z 235.586,A -85,B 0,C 180,E1 -3608.9,E2 -3608.9} C_VEL
LIN {X 0,Y 545.077,Z 235.59,A -85,B 0,C 180,E1 -3611.905,E2 -3611.905} C_VEL
LIN {X 0,Y 545.085,Z 235.586,A -85,B 0,C 180,E1 -3614.944,E2 -3614.944} C_VEL
LIN {X 0,Y 545.081,Z 235.586,A -85,B 0,C 180,E1 -3618.026,E2 -3618.026} C_VEL
LIN {X 0,Y 545.096,Z 235.588,A -85,B 0,C 180,E1 -3620.372,E2 -3620.372} C_VEL
LIN {X 0,Y 545.075,Z 235.587,A -85,B 0,C 180,E1 -3623.56,E2 -3623.56} C_VEL
LIN {X 0,Y 545.058,Z 235.588,A -85,B 0,C 180,E1 -3626.827,E2 -3626.827} C_VEL
LIN {X 0,Y 545.046,Z 235.595,A -85,B 0,C 180,E1 -3629.34,E2 -3629.34} C_VEL
LIN {X 0,Y 545.059,Z 235.589,A -85,B 0,C 180,E1 -3631.915,E2 -3631.915} C_VEL
LIN {X 0,Y 545.064,Z 235.591,A -85,B 0,C 180,E1 -3634.564,E2 -3634.564} C_VEL
LIN {X 0,Y 545.03,Z 235.593,A -85,B 0,C 180,E1 -3637.305,E2 -3637.305} C_VEL
LIN {X 0,Y 545.062,Z 235.587,A -85,B 0,C 180,E1 -3640.143,E2 -3640.143} C_VEL
LIN {X 0,Y 545.048,Z 235.593,A -85,B 0,C 180,E1 -3643.11,E2 -3643.11} C_VEL
LIN {X 0,Y 545.052,Z 235.595,A -85,B 0,C 180,E1 -3646.226,E2 -3646.226} C_VEL
LIN {X 0,Y 545.084,Z 235.586,A -85,B 0,C 180,E1 -3648.885,E2 -3648.885} C_VEL
LIN {X 0,Y 545.048,Z 235.594,A -85,B 0,C 180,E1 -3651.865,E2 -3651.865} C_VEL
LIN {X 0,Y 545.111,Z 235.7,A -85,B 0,C 180,E1 -3653.136,E2 -3653.136} C_VEL
LIN {X 0,Y 545.521,Z 240.122,A -85,B 0,C 180,E1 -3655.019,E2 -3655.019} C_VEL
LIN {X 0,Y 545.406,Z 247.857,A -85,B 0,C 180,E1 -3658.108,E2 -3658.108} C_VEL
LIN {X 0,Y 545.22,Z 256.057,A -85,B 0,C 180,E1 -3661.228,E2 -3661.228} C_VEL
LIN {X 0,Y 545.116,Z 264.924,A -85,B 0,C 180,E1 -3664.487,E2 -3664.487} C_VEL
LIN {X 0,Y 545.018,Z 272.591,A -85,B 0,C 180,E1 -3667.241,E2 -3667.241} C_VEL
LIN {X 0,Y 544.938,Z 279.31,A -85,B 0,C 180,E1 -3669.622,E2 -3669.622} C_VEL
LIN {X 0,Y 544.877,Z 287.333,A -85,B 0,C 180,E1 -3672.394,E2 -3672.394} C_VEL
LIN {X 0,Y 544.823,Z 296.044,A -85,B 0,C 180,E1 -3675.346,E2 -3675.346} C_VEL
LIN {X 0,Y 544.757,Z 300.466,A -85,B 0,C 180,E1 -3676.833,E2 -3676.833} C_VEL
LIN {X 0,Y 546.167,Z 310.346,A -85,B 0,C 180,E1 -3677.081,E2 -3677.081} C_VEL
LIN {X 0,Y 546.019,Z 322.47,A -85,B 0,C 180,E1 -3677.455,E2 -3677.455} C_VEL
LIN {X 0,Y 545.779,Z 333.486,A -85,B 0,C 180,E1 -3677.921,E2 -3677.921} C_VEL
LIN {X 0,Y 545.585,Z 344.158,A -85,B 0,C 180,E1 -3678.505,E2 -3678.505} C_VEL
LIN {X 0,Y 545.424,Z 354.741,A -85,B 0,C 180,E1 -3679.232,E2 -3679.232} C_VEL
LIN {X 0,Y 545.225,Z 365.596,A -85,B 0,C 180,E1 -3680.166,E2 -3680.166} C_VEL
LIN {X 0,Y 545.051,Z 374.411,A -85,B 0,C 180,E1 -3681.099,E2 -3681.099} C_VEL
LIN {X 0,Y 544.896,Z 383.003,A -85,B 0,C 180,E1 -3682.217,E2 -3682.217} C_VEL
LIN {X 0,Y 544.745,Z 390.348,A -85,B 0,C 180,E1 -3683.421,E2 -3683.421} C_VEL
LIN {X 0,Y 544.741,Z 395.365,A -85,B 0,C 180,E1 -3684.447,E2 -3684.447} C_VEL
LIN {X 0,Y 544.66,Z 399.676,A -85,B 0,C 180,E1 -3685.56,E2 -3685.56} C_VEL
LIN {X 0,Y 544.669,Z 401.958,A -85,B 0,C 180,E1 -3686.301,E2 -3686.301} C_VEL
LIN {X 0,Y 544.65,Z 403.807,A -85,B 0,C 180,E1 -3687.041,E2 -3687.041} C_VEL
LIN {X 0,Y 544.546,Z 406.182,A -85,B 0,C 180,E1 -3688.521,E2 -3688.521} C_VEL
LIN {X 0,Y 544.541,Z 407,A -85,B 0,C 180,E1 -3690,E2 -3690} C_VEL
LIN {X 0,Y 544.546,Z 406.184,A -85,B 0,C 180,E1 -3691.479,E2 -3691.479} C_VEL
LIN {X 0,Y 544.65,Z 403.81,A -85,B 0,C 180,E1 -3692.959,E2 -3692.959} C_VEL
LIN {X 0,Y 544.684,Z 400.895,A -85,B 0,C 180,E1 -3694.069,E2 -3694.069} C_VEL
LIN {X 0,Y 544.653,Z 396.948,A -85,B 0,C 180,E1 -3695.182,E2 -3695.182} C_VEL
LIN {X 0,Y 544.73,Z 391.642,A -85,B 0,C 180,E1 -3696.34,E2 -3696.34} C_VEL
LIN {X 0,Y 544.836,Z 385.467,A -85,B 0,C 180,E1 -3697.411,E2 -3697.411} C_VEL
LIN {X 0,Y 545.006,Z 377.477,A -85,B 0,C 180,E1 -3698.528,E2 -3698.528} C_VEL
LIN {X 0,Y 545.142,Z 369.333,A -85,B 0,C 180,E1 -3699.461,E2 -3699.461} C_VEL
LIN {X 0,Y 545.369,Z 359.397,A -85,B 0,C 180,E1 -3700.394,E2 -3700.394} C_VEL
LIN {X 0,Y 545.5,Z 349.592,A -85,B 0,C 180,E1 -3701.143,E2 -3701.143} C_VEL
LIN {X 0,Y 545.69,Z 338.624,A -85,B 0,C 180,E1 -3701.814,E2 -3701.814} C_VEL
LIN {X 0,Y 545.875,Z 326.101,A -85,B 0,C 180,E1 -3702.407,E2 -3702.407} C_VEL
LIN {X 0,Y 546.104,Z 313.087,A -85,B 0,C 180,E1 -3702.85,E2 -3702.85} C_VEL
LIN {X 0,Y 545.907,Z 307.501,A -85,B 0,C 180,E1 -3702.997,E2 -3702.997} C_VEL
LIN {X 0,Y 544.758,Z 300.467,A -85,B 0,C 180,E1 -3703.167,E2 -3703.167} C_VEL
LIN {X 0,Y 544.827,Z 292.896,A -85,B 0,C 180,E1 -3705.717,E2 -3705.717} C_VEL
LIN {X 0,Y 544.859,Z 284.945,A -85,B 0,C 180,E1 -3708.422,E2 -3708.422} C_VEL
LIN {X 0,Y 544.987,Z 277.082,A -85,B 0,C 180,E1 -3711.167,E2 -3711.167} C_VEL
LIN {X 0,Y 545.093,Z 268.094,A -85,B 0,C 180,E1 -3714.367,E2 -3714.367} C_VEL
LIN {X 0,Y 545.131,Z 260.349,A -85,B 0,C 180,E1 -3717.18,E2 -3717.18} C_VEL
LIN {X 0,Y 545.286,Z 253.451,A -85,B 0,C 180,E1 -3719.75,E2 -3719.75} C_VEL
LIN {X 0,Y 545.431,Z 245.622,A -85,B 0,C 180,E1 -3722.764,E2 -3722.764} C_VEL
LIN {X 0,Y 545.535,Z 239.03,A -85,B 0,C 180,E1 -3725.431,E2 -3725.431} C_VEL
LIN {X 0,Y 545.076,Z 235.593,A -85,B 0,C 180,E1 -3726.926,E2 -3726.926} C_VEL
LIN {X 0,Y 545.066,Z 235.594,A -85,B 0,C 180,E1 -3730.143,E2 -3730.143} C_VEL
LIN {X 0,Y 545.081,Z 235.586,A -85,B 0,C 180,E1 -3733.107,E2 -3733.107} C_VEL
LIN {X 0,Y 545.051,Z 235.589,A -85,B 0,C 180,E1 -3736.226,E2 -3736.226} C_VEL
LIN {X 0,Y 545.029,Z 235.597,A -85,B 0,C 180,E1 -3738.88,E2 -3738.88} C_VEL
LIN {X 0,Y 545.045,Z 235.59,A -85,B 0,C 180,E1 -3741.762,E2 -3741.762} C_VEL
LIN {X 0,Y 545.032,Z 235.593,A -85,B 0,C 180,E1 -3744.531,E2 -3744.531} C_VEL
LIN {X 0,Y 545.083,Z 235.589,A -85,B 0,C 180,E1 -3747.212,E2 -3747.212} C_VEL
LIN {X 0,Y 545.064,Z 235.588,A -85,B 0,C 180,E1 -3749.81,E2 -3749.81} C_VEL
LIN {X 0,Y 545.048,Z 235.593,A -85,B 0,C 180,E1 -3752.342,E2 -3752.342} C_VEL
LIN {X 0,Y 545.041,Z 235.59,A -85,B 0,C 180,E1 -3754.817,E2 -3754.817} C_VEL
LIN {X 0,Y 545.035,Z 235.592,A -85,B 0,C 180,E1 -3757.242,E2 -3757.242} C_VEL
LIN {X 0,Y 545.119,Z 235.581,A -85,B 0,C 180,E1 -3760.415,E2 -3760.415} C_VEL
LIN {X 0,Y 545.071,Z 235.587,A -85,B 0,C 180,E1 -3763.521,E2 -3763.521} C_VEL
LIN {X 0,Y 545.09,Z 235.586,A -85,B 0,C 180,E1 -3765.82,E2 -3765.82} C_VEL
LIN {X 0,Y 545.112,Z 235.581,A -85,B 0,C 180,E1 -3768.849,E2 -3768.849} C_VEL
LIN {X 0,Y 545.088,Z 235.586,A -85,B 0,C 180,E1 -3771.846,E2 -3771.846} C_VEL
LIN {X 0,Y 545.168,Z 235.574,A -85,B 0,C 180,E1 -3774.08,E2 -3774.08} C_VEL
LIN {X 0,Y 545.173,Z 235.576,A -85,B 0,C 180,E1 -3777.044,E2 -3777.044} C_VEL
LIN {X 0,Y 545.204,Z 235.575,A -85,B 0,C 180,E1 -3780,E2 -3780} C_VEL
LIN {X 0,Y 545.155,Z 235.577,A -85,B 0,C 180,E1 -3782.956,E2 -3782.956} C_VEL
LIN {X 0,Y 545.133,Z 235.578,A -85,B 0,C 180,E1 -3785.92,E2 -3785.92} C_VEL
LIN {X 0,Y 545.113,Z 235.584,A -85,B 0,C 180,E1 -3788.9,E2 -3788.9} C_VEL
LIN {X 0,Y 545.138,Z 235.583,A -85,B 0,C 180,E1 -3791.904,E2 -3791.904} C_VEL
LIN {X 0,Y 545.083,Z 235.587,A -85,B 0,C 180,E1 -3794.944,E2 -3794.944} C_VEL
LIN {X 0,Y 545.057,Z 235.588,A -85,B 0,C 180,E1 -3798.027,E2 -3798.027} C_VEL
LIN {X 0,Y 545.093,Z 235.587,A -85,B 0,C 180,E1 -3800.372,E2 -3800.372} C_VEL
LIN {X 0,Y 545.082,Z 235.587,A -85,B 0,C 180,E1 -3803.559,E2 -3803.559} C_VEL
LIN {X 0,Y 545.083,Z 235.588,A -85,B 0,C 180,E1 -3806.001,E2 -3806.001} C_VEL
LIN {X 0,Y 545.071,Z 235.589,A -85,B 0,C 180,E1 -3808.744,E2 -3808.744} C_VEL
LIN {X 0,Y 545.059,Z 235.588,A -85,B 0,C 180,E1 -3811.679,E2 -3811.679} C_VEL
LIN {X 0,Y 545.057,Z 235.59,A -85,B 0,C 180,E1 -3814.565,E2 -3814.565} C_VEL
LIN {X 0,Y 545.06,Z 235.587,A -85,B 0,C 180,E1 -3816.988,E2 -3816.988} C_VEL
LIN {X 0,Y 544.353,Z 235.68,A -85,B 0,C 180,E1 -3817.604,E2 -3817.604} C_VEL
LIN {X 0,Y 541.49,Z 236.035,A -85,B 0,C 180,E1 -3818.605,E2 -3818.605} C_VEL
LIN {X 0,Y 539.104,Z 236.335,A -85,B 0,C 180,E1 -3819.411,E2 -3819.411} C_VEL
LIN {X 0,Y 538.094,Z 236.457,A -85,B 0,C 180,E1 -3820.033,E2 -3820.033} C_VEL
LIN {X 0,Y 538.018,Z 236.465,A -85,B 0,C 180,E1 -3820.244,E2 -3820.244} C_VEL
LIN {X 0,Y 537.982,Z 236.475,A -85,B 0,C 180,E1 -3822.982,E2 -3822.982} C_VEL
LIN {X 0,Y 537.997,Z 236.471,A -85,B 0,C 180,E1 -3825.929,E2 -3825.929} C_VEL
LIN {X 0,Y 538.003,Z 236.468,A -85,B 0,C 180,E1 -3829.259,E2 -3829.259} C_VEL
LIN {X 0,Y 537.994,Z 236.468,A -85,B 0,C 180,E1 -3832.122,E2 -3832.122} C_VEL
LIN {X 0,Y 537.954,Z 236.474,A -85,B 0,C 180,E1 -3834.095,E2 -3834.095} C_VEL
LIN {X 0,Y 537.93,Z 236.796,A -85,B 0,C 180,E1 -3834.91,E2 -3834.91} C_VEL
LIN {X 0,Y 537.888,Z 240.964,A -85,B 0,C 180,E1 -3837.608,E2 -3837.608} C_VEL
LIN {X 0,Y 537.848,Z 245.076,A -85,B 0,C 180,E1 -3840.229,E2 -3840.229} C_VEL
LIN {X 0,Y 537.788,Z 249.162,A -85,B 0,C 180,E1 -3842.781,E2 -3842.781} C_VEL
LIN {X 0,Y 537.774,Z 253.238,A -85,B 0,C 180,E1 -3845.279,E2 -3845.279} C_VEL
LIN {X 0,Y 537.718,Z 258.672,A -85,B 0,C 180,E1 -3848.533,E2 -3848.533} C_VEL
LIN {X 0,Y 537.65,Z 262.74,A -85,B 0,C 180,E1 -3850.926,E2 -3850.926} C_VEL
LIN {X 0,Y 537.633,Z 266.811,A -85,B 0,C 180,E1 -3853.287,E2 -3853.287} C_VEL
LIN {X 0,Y 537.619,Z 270.87,A -85,B 0,C 180,E1 -3855.619,E2 -3855.619} C_VEL
LIN {X 0,Y 537.573,Z 272.833,A -85,B 0,C 180,E1 -3856.738,E2 -3856.738} C_VEL
LIN {X 0,Y 539.204,Z 283.441,A -85,B 0,C 180,E1 -3857.031,E2 -3857.031} C_VEL
LIN {X 0,Y 538.982,Z 296.396,A -85,B 0,C 180,E1 -3857.48,E2 -3857.48} C_VEL
LIN {X 0,Y 538.816,Z 308.899,A -85,B 0,C 180,E1 -3858.082,E2 -3858.082} C_VEL
LIN {X 0,Y 538.565,Z 320.462,A -85,B 0,C 180,E1 -3858.807,E2 -3858.807} C_VEL
LIN {X 0,Y 538.298,Z 331.163,A -85,B 0,C 180,E1 -3859.658,E2 -3859.658} C_VEL
LIN {X 0,Y 538.108,Z 340.789,A -85,B 0,C 180,E1 -3860.604,E2 -3860.604} C_VEL
LIN {X 0,Y 537.937,Z 348.673,A -85,B 0,C 180,E1 -3861.548,E2 -3861.548} C_VEL
LIN {X 0,Y 537.76,Z 356.385,A -85,B 0,C 180,E1 -3862.679,E2 -3862.679} C_VEL
LIN {X 0,Y 537.694,Z 363.462,A -85,B 0,C 180,E1 -3863.998,E2 -3863.998} C_VEL
LIN {X 0,Y 537.54,Z 368.201,A -85,B 0,C 180,E1 -3865.125,E2 -3865.125} C_VEL
LIN {X 0,Y 537.591,Z 371.833,A -85,B 0,C 180,E1 -3866.252,E2 -3866.252} C_VEL
LIN {X 0,Y 537.551,Z 373.71,A -85,B 0,C 180,E1 -3867.002,E2 -3867.002} C_VEL
LIN {X 0,Y 537.489,Z 375.128,A -85,B 0,C 180,E1 -3867.752,E2 -3867.752} C_VEL
LIN {X 0,Y 537.442,Z 376.757,A -85,B 0,C 180,E1 -3869.251,E2 -3869.251} C_VEL
LIN {X 0,Y 537.442,Z 376.996,A -85,B 0,C 180,E1 -3870,E2 -3870} C_VEL
LIN {X 0,Y 537.442,Z 376.814,A -85,B 0,C 180,E1 -3870.749,E2 -3870.749} C_VEL
LIN {X 0,Y 537.489,Z 375.26,A -85,B 0,C 180,E1 -3872.248,E2 -3872.248} C_VEL
LIN {X 0,Y 537.552,Z 373.899,A -85,B 0,C 180,E1 -3872.998,E2 -3872.998} C_VEL
LIN {X 0,Y 537.603,Z 371.021,A -85,B 0,C 180,E1 -3874.123,E2 -3874.123} C_VEL
LIN {X 0,Y 537.587,Z 367.119,A -85,B 0,C 180,E1 -3875.251,E2 -3875.251} C_VEL
LIN {X 0,Y 537.639,Z 362.368,A -85,B 0,C 180,E1 -3876.321,E2 -3876.321} C_VEL
LIN {X 0,Y 537.79,Z 355.786,A -85,B 0,C 180,E1 -3877.509,E2 -3877.509} C_VEL
LIN {X 0,Y 537.952,Z 347.897,A -85,B 0,C 180,E1 -3878.641,E2 -3878.641} C_VEL
LIN {X 0,Y 538.14,Z 338.082,A -85,B 0,C 180,E1 -3879.775,E2 -3879.775} C_VEL
LIN {X 0,Y 538.366,Z 327.791,A -85,B 0,C 180,E1 -3880.721,E2 -3880.721} C_VEL
LIN {X 0,Y 538.619,Z 316.844,A -85,B 0,C 180,E1 -3881.528,E2 -3881.528} C_VEL
LIN {X 0,Y 538.846,Z 306.441,A -85,B 0,C 180,E1 -3882.141,E2 -3882.141} C_VEL
LIN {X 0,Y 539.05,Z 293.925,A -85,B 0,C 180,E1 -3882.71,E2 -3882.71} C_VEL
LIN {X 0,Y 539.078,Z 281.403,A -85,B 0,C 180,E1 -3883.116,E2 -3883.116} C_VEL
LIN {X 0,Y 537.566,Z 272.776,A -85,B 0,C 180,E1 -3883.37,E2 -3883.37} C_VEL
LIN {X 0,Y 537.594,Z 268.33,A -85,B 0,C 180,E1 -3885.934,E2 -3885.934} C_VEL
LIN {X 0,Y 537.613,Z 264.285,A -85,B 0,C 180,E1 -3888.285,E2 -3888.285} C_VEL
LIN {X 0,Y 537.662,Z 260.182,A -85,B 0,C 180,E1 -3890.667,E2 -3890.667} C_VEL
LIN {X 0,Y 537.711,Z 256.11,A -85,B 0,C 180,E1 -3893.086,E2 -3893.086} C_VEL
LIN {X 0,Y 537.763,Z 251.925,A -85,B 0,C 180,E1 -3895.609,E2 -3895.609} C_VEL
LIN {X 0,Y 537.822,Z 247.949,A -85,B 0,C 180,E1 -3898.062,E2 -3898.062} C_VEL
LIN {X 0,Y 537.843,Z 243.859,A -85,B 0,C 180,E1 -3900.638,E2 -3900.638} C_VEL
LIN {X 0,Y 537.931,Z 239.732,A -85,B 0,C 180,E1 -3903.28,E2 -3903.28} C_VEL
LIN {X 0,Y 537.926,Z 236.94,A -85,B 0,C 180,E1 -3905.09,E2 -3905.09} C_VEL
LIN {X 0,Y 537.963,Z 236.472,A -85,B 0,C 180,E1 -3906.007,E2 -3906.007} C_VEL
LIN {X 0,Y 538.016,Z 236.469,A -85,B 0,C 180,E1 -3908.831,E2 -3908.831} C_VEL
LIN {X 0,Y 537.991,Z 236.471,A -85,B 0,C 180,E1 -3911.874,E2 -3911.874} C_VEL
LIN {X 0,Y 537.993,Z 236.471,A -85,B 0,C 180,E1 -3915.136,E2 -3915.136} C_VEL
LIN {X 0,Y 538.027,Z 236.465,A -85,B 0,C 180,E1 -3918.226,E2 -3918.226} C_VEL
LIN {X 0,Y 538.015,Z 236.466,A -85,B 0,C 180,E1 -3921.169,E2 -3921.169} C_VEL
LIN {X 0,Y 537.998,Z 236.474,A -85,B 0,C 180,E1 -3924.089,E2 -3924.089} C_VEL
LIN {X 0,Y 538.034,Z 236.463,A -85,B 0,C 180,E1 -3926.727,E2 -3926.727} C_VEL
LIN {X 0,Y 538.005,Z 236.47,A -85,B 0,C 180,E1 -3929.561,E2 -3929.561} C_VEL
LIN {X 0,Y 538.03,Z 236.464,A -85,B 0,C 180,E1 -3931.949,E2 -3931.949} C_VEL
LIN {X 0,Y 538.076,Z 236.462,A -85,B 0,C 180,E1 -3934.467,E2 -3934.467} C_VEL
LIN {X 0,Y 537.997,Z 236.474,A -85,B 0,C 180,E1 -3937.738,E2 -3937.738} C_VEL
LIN {X 0,Y 538.084,Z 236.456,A -85,B 0,C 180,E1 -3940.148,E2 -3940.148} C_VEL
LIN {X 0,Y 537.989,Z 236.471,A -85,B 0,C 180,E1 -3943.298,E2 -3943.298} C_VEL
LIN {X 0,Y 538.06,Z 236.461,A -85,B 0,C 180,E1 -3945.63,E2 -3945.63} C_VEL
LIN {X 0,Y 538.081,Z 236.458,A -85,B 0,C 180,E1 -3948.702,E2 -3948.702} C_VEL
LIN {X 0,Y 538.064,Z 236.462,A -85,B 0,C 180,E1 -3951.739,E2 -3951.739} C_VEL
LIN {X 0,Y 538.149,Z 236.452,A -85,B 0,C 180,E1 -3954.755,E2 -3954.755} C_VEL
LIN {X 0,Y 538.156,Z 236.448,A -85,B 0,C 180,E1 -3957.755,E2 -3957.755} C_VEL
LIN {X 0,Y 538.183,Z 236.445,A -85,B 0,C 180,E1 -3960.748,E2 -3960.748} C_VEL
LIN {X 0,Y 538.141,Z 236.452,A -85,B 0,C 180,E1 -3962.994,E2 -3962.994} C_VEL
LIN {X 0,Y 538.12,Z 236.452,A -85,B 0,C 180,E1 -3965.997,E2 -3965.997} C_VEL
LIN {X 0,Y 538.055,Z 236.462,A -85,B 0,C 180,E1 -3968.261,E2 -3968.261} C_VEL
LIN {X 0,Y 538.045,Z 236.463,A -85,B 0,C 180,E1 -3971.575,E2 -3971.575} C_VEL
LIN {X 0,Y 538.061,Z 236.461,A -85,B 0,C 180,E1 -3974.856,E2 -3974.856} C_VEL
LIN {X 0,Y 538.064,Z 236.462,A -85,B 0,C 180,E1 -3977.54,E2 -3977.54} C_VEL
LIN {X 0,Y 538.041,Z 236.467,A -85,B 0,C 180,E1 -3980.651,E2 -3980.651} C_VEL
LIN {X 0,Y 538.009,Z 236.471,A -85,B 0,C 180,E1 -3983.878,E2 -3983.878} C_VEL
LIN {X 0,Y 537.992,Z 236.468,A -85,B 0,C 180,E1 -3986.369,E2 -3986.369} C_VEL
LIN {X 0,Y 538.033,Z 236.467,A -85,B 0,C 180,E1 -3988.933,E2 -3988.933} C_VEL
LIN {X 0,Y 538.014,Z 236.466,A -85,B 0,C 180,E1 -3991.887,E2 -3991.887} C_VEL
LIN {X 0,Y 538.014,Z 236.469,A -85,B 0,C 180,E1 -3994.617,E2 -3994.617} C_VEL
LIN {X 0,Y 538,Z 236.468,A -85,B 0,C 180,E1 -3997.169,E2 -3997.169} C_VEL
LIN {X 0,Y 538.008,Z 236.468,A -85,B 0,C 180,E1 -3999.798,E2 -3999.798} C_VEL
LIN {X 0,Y 538.001,Z 236.473,A -85,B 0,C 180,E1 -4002.984,E2 -4002.984} C_VEL
LIN {X 0,Y 538.021,Z 236.468,A -85,B 0,C 180,E1 -4005.927,E2 -4005.927} C_VEL
LIN {X 0,Y 538.033,Z 236.468,A -85,B 0,C 180,E1 -4008.227,E2 -4008.227} C_VEL
LIN {X 0,Y 538.012,Z 236.47,A -85,B 0,C 180,E1 -4011.169,E2 -4011.169} C_VEL
LIN {X 0,Y 538.09,Z 236.603,A -85,B 0,C 180,E1 -4012.982,E2 -4012.982} C_VEL
LIN {X 0,Y 538.534,Z 241.169,A -85,B 0,C 180,E1 -4014.955,E2 -4014.955} C_VEL
LIN {X 0,Y 538.43,Z 247.788,A -85,B 0,C 180,E1 -4017.645,E2 -4017.645} C_VEL
LIN {X 0,Y 538.265,Z 255.611,A -85,B 0,C 180,E1 -4020.684,E2 -4020.684} C_VEL
LIN {X 0,Y 538.115,Z 263.473,A -85,B 0,C 180,E1 -4023.637,E2 -4023.637} C_VEL
LIN {X 0,Y 537.992,Z 271.367,A -85,B 0,C 180,E1 -4026.524,E2 -4026.524} C_VEL
LIN {X 0,Y 537.898,Z 279.212,A -85,B 0,C 180,E1 -4029.343,E2 -4029.343} C_VEL
LIN {X 0,Y 537.818,Z 287.062,A -85,B 0,C 180,E1 -4032.116,E2 -4032.116} C_VEL
LIN {X 0,Y 537.735,Z 296.257,A -85,B 0,C 180,E1 -4035.275,E2 -4035.275} C_VEL
LIN {X 0,Y 537.67,Z 300.311,A -85,B 0,C 180,E1 -4036.656,E2 -4036.656} C_VEL
LIN {X 0,Y 539.22,Z 311.077,A -85,B 0,C 180,E1 -4036.935,E2 -4036.935} C_VEL
LIN {X 0,Y 539.036,Z 323.606,A -85,B 0,C 180,E1 -4037.338,E2 -4037.338} C_VEL
LIN {X 0,Y 538.812,Z 335.263,A -85,B 0,C 180,E1 -4037.858,E2 -4037.858} C_VEL
LIN {X 0,Y 538.581,Z 346.045,A -85,B 0,C 180,E1 -4038.482,E2 -4038.482} C_VEL
LIN {X 0,Y 538.373,Z 357.013,A -85,B 0,C 180,E1 -4039.279,E2 -4039.279} C_VEL
LIN {X 0,Y 538.135,Z 367.501,A -85,B 0,C 180,E1 -4040.225,E2 -4040.225} C_VEL
LIN {X 0,Y 537.974,Z 375.989,A -85,B 0,C 180,E1 -4041.17,E2 -4041.17} C_VEL
LIN {X 0,Y 537.817,Z 384.234,A -85,B 0,C 180,E1 -4042.302,E2 -4042.302} C_VEL
LIN {X 0,Y 537.683,Z 390.749,A -85,B 0,C 180,E1 -4043.409,E2 -4043.409} C_VEL
LIN {X 0,Y 537.676,Z 395.366,A -85,B 0,C 180,E1 -4044.374,E2 -4044.374} C_VEL
LIN {X 0,Y 537.557,Z 399.676,A -85,B 0,C 180,E1 -4045.501,E2 -4045.501} C_VEL
LIN {X 0,Y 537.591,Z 401.957,A -85,B 0,C 180,E1 -4046.252,E2 -4046.252} C_VEL
LIN {X 0,Y 537.551,Z 403.806,A -85,B 0,C 180,E1 -4047.002,E2 -4047.002} C_VEL
LIN {X 0,Y 537.451,Z 406.182,A -85,B 0,C 180,E1 -4048.501,E2 -4048.501} C_VEL
LIN {X 0,Y 537.442,Z 407,A -85,B 0,C 180,E1 -4050,E2 -4050} C_VEL
LIN {X 0,Y 537.451,Z 406.183,A -85,B 0,C 180,E1 -4051.499,E2 -4051.499} C_VEL
LIN {X 0,Y 537.551,Z 403.81,A -85,B 0,C 180,E1 -4052.998,E2 -4052.998} C_VEL
LIN {X 0,Y 537.603,Z 400.895,A -85,B 0,C 180,E1 -4054.123,E2 -4054.123} C_VEL
LIN {X 0,Y 537.587,Z 396.948,A -85,B 0,C 180,E1 -4055.251,E2 -4055.251} C_VEL
LIN {X 0,Y 537.644,Z 392.124,A -85,B 0,C 180,E1 -4056.326,E2 -4056.326} C_VEL
LIN {X 0,Y 537.791,Z 385.466,A -85,B 0,C 180,E1 -4057.509,E2 -4057.509} C_VEL
LIN {X 0,Y 537.972,Z 377.477,A -85,B 0,C 180,E1 -4058.64,E2 -4058.64} C_VEL
LIN {X 0,Y 538.118,Z 369.304,A -85,B 0,C 180,E1 -4059.585,E2 -4059.585} C_VEL
LIN {X 0,Y 538.372,Z 359.33,A -85,B 0,C 180,E1 -4060.53,E2 -4060.53} C_VEL
LIN {X 0,Y 538.531,Z 349.492,A -85,B 0,C 180,E1 -4061.289,E2 -4061.289} C_VEL
LIN {X 0,Y 538.715,Z 338.459,A -85,B 0,C 180,E1 -4061.971,E2 -4061.971} C_VEL
LIN {X 0,Y 538.945,Z 325.94,A -85,B 0,C 180,E1 -4062.569,E2 -4062.569} C_VEL
LIN {X 0,Y 539.179,Z 312.904,A -85,B 0,C 180,E1 -4063.018,E2 -4063.018} C_VEL
LIN {X 0,Y 539.006,Z 308.321,A -85,B 0,C 180,E1 -4063.142,E2 -4063.142} C_VEL
LIN {X 0,Y 537.67,Z 300.312,A -85,B 0,C 180,E1 -4063.343,E2 -4063.343} C_VEL
LIN {X 0,Y 537.771,Z 291.606,A -85,B 0,C 180,E1 -4066.319,E2 -4066.319} C_VEL
LIN {X 0,Y 537.845,Z 283.65,A -85,B 0,C 180,E1 -4069.067,E2 -4069.067} C_VEL
LIN {X 0,Y 537.963,Z 275.614,A -85,B 0,C 180,E1 -4071.943,E2 -4071.943} C_VEL
LIN {X 0,Y 538.029,Z 267.979,A -85,B 0,C 180,E1 -4074.708,E2 -4074.708} C_VEL
LIN {X 0,Y 538.101,Z 260.799,A -85,B 0,C 180,E1 -4077.36,E2 -4077.36} C_VEL
LIN {X 0,Y 538.264,Z 254.482,A -85,B 0,C 180,E1 -4079.746,E2 -4079.746} C_VEL
LIN {X 0,Y 538.43,Z 247.78,A -85,B 0,C 180,E1 -4082.355,E2 -4082.355} C_VEL
LIN {X 0,Y 538.531,Z 241.167,A -85,B 0,C 180,E1 -4085.045,E2 -4085.045} C_VEL
LIN {X 0,Y 538.06,Z 236.608,A -85,B 0,C 180,E1 -4087.017,E2 -4087.017} C_VEL
LIN {X 0,Y 538.023,Z 236.469,A -85,B 0,C 180,E1 -4089.797,E2 -4089.797} C_VEL
LIN {X 0,Y 538.021,Z 236.465,A -85,B 0,C 180,E1 -4092.786,E2 -4092.786} C_VEL
LIN {X 0,Y 538.021,Z 236.466,A -85,B 0,C 180,E1 -4095.927,E2 -4095.927} C_VEL
LIN {X 0,Y 538.003,Z 236.468,A -85,B 0,C 180,E1 -4099.22,E2 -4099.22} C_VEL
LIN {X 0,Y 537.986,Z 236.473,A -85,B 0,C 180,E1 -4102.122,E2 -4102.122} C_VEL
LIN {X 0,Y 537.997,Z 236.468,A -85,B 0,C 180,E1 -4104.915,E2 -4104.915} C_VEL
LIN {X 0,Y 538.029,Z 236.469,A -85,B 0,C 180,E1 -4107.618,E2 -4107.618} C_VEL
LIN {X 0,Y 538.014,Z 236.467,A -85,B 0,C 180,E1 -4110.239,E2 -4110.239} C_VEL
LIN {X 0,Y 538.016,Z 236.469,A -85,B 0,C 180,E1 -4112.793,E2 -4112.793} C_VEL
LIN {X 0,Y 537.985,Z 236.468,A -85,B 0,C 180,E1 -4115.289,E2 -4115.289} C_VEL
LIN {X 0,Y 538.017,Z 236.468,A -85,B 0,C 180,E1 -4118.042,E2 -4118.042} C_VEL
LIN {X 0,Y 538.036,Z 236.467,A -85,B 0,C 180,E1 -4120.94,E2 -4120.94} C_VEL
LIN {X 0,Y 538.024,Z 236.467,A -85,B 0,C 180,E1 -4123.299,E2 -4123.299} C_VEL
LIN {X 0,Y 538.061,Z 236.46,A -85,B 0,C 180,E1 -4125.631,E2 -4125.631} C_VEL
LIN {X 0,Y 538.073,Z 236.458,A -85,B 0,C 180,E1 -4128.701,E2 -4128.701} C_VEL
LIN {X 0,Y 538.053,Z 236.463,A -85,B 0,C 180,E1 -4131.739,E2 -4131.739} C_VEL
LIN {X 0,Y 538.119,Z 236.452,A -85,B 0,C 180,E1 -4134.003,E2 -4134.003} C_VEL
LIN {X 0,Y 538.14,Z 236.452,A -85,B 0,C 180,E1 -4137.006,E2 -4137.006} C_VEL
LIN {X 0,Y 538.175,Z 236.45,A -85,B 0,C 180,E1 -4140,E2 -4140} C_VEL
LIN {X 0,Y 538.123,Z 236.454,A -85,B 0,C 180,E1 -4142.995,E2 -4142.995} C_VEL
LIN {X 0,Y 538.089,Z 236.455,A -85,B 0,C 180,E1 -4145.998,E2 -4145.998} C_VEL
LIN {X 0,Y 538.066,Z 236.461,A -85,B 0,C 180,E1 -4149.018,E2 -4149.018} C_VEL
LIN {X 0,Y 538.086,Z 236.462,A -85,B 0,C 180,E1 -4152.063,E2 -4152.063} C_VEL
LIN {X 0,Y 538.042,Z 236.466,A -85,B 0,C 180,E1 -4155.144,E2 -4155.144} C_VEL
LIN {X 0,Y 538.011,Z 236.467,A -85,B 0,C 180,E1 -4158.271,E2 -4158.271} C_VEL
LIN {X 0,Y 538.039,Z 236.467,A -85,B 0,C 180,E1 -4160.652,E2 -4160.652} C_VEL
LIN {X 0,Y 538.005,Z 236.471,A -85,B 0,C 180,E1 -4163.888,E2 -4163.888} C_VEL
LIN {X 0,Y 538.045,Z 236.463,A -85,B 0,C 180,E1 -4166.367,E2 -4166.367} C_VEL
LIN {X 0,Y 538.032,Z 236.468,A -85,B 0,C 180,E1 -4168.933,E2 -4168.933} C_VEL
LIN {X 0,Y 538.011,Z 236.466,A -85,B 0,C 180,E1 -4171.887,E2 -4171.887} C_VEL
LIN {X 0,Y 538.006,Z 236.468,A -85,B 0,C 180,E1 -4174.616,E2 -4174.616} C_VEL
LIN {X 0,Y 538.002,Z 236.467,A -85,B 0,C 180,E1 -4177.169,E2 -4177.169} C_VEL
LIN {X 0,Y 538.018,Z 236.465,A -85,B 0,C 180,E1 -4180.244,E2 -4180.244} C_VEL
LIN {X 0,Y 537.366,Z 236.55,A -85,B 0,C 180,E1 -4180.869,E2 -4180.869} C_VEL
LIN {X 0,Y 534.505,Z 236.905,A -85,B 0,C 180,E1 -4181.883,E2 -4181.883} C_VEL
LIN {X 0,Y 532.074,Z 237.21,A -85,B 0,C 180,E1 -4182.7,E2 -4182.7} C_VEL
LIN {X 0,Y 531.025,Z 237.339,A -85,B 0,C 180,E1 -4183.331,E2 -4183.331} C_VEL
LIN {X 0,Y 530.937,Z 237.348,A -85,B 0,C 180,E1 -4183.545,E2 -4183.545} C_VEL
LIN {X 0,Y 530.925,Z 237.352,A -85,B 0,C 180,E1 -4186.501,E2 -4186.501} C_VEL
LIN {X 0,Y 530.953,Z 237.35,A -85,B 0,C 180,E1 -4189.564,E2 -4189.564} C_VEL
LIN {X 0,Y 530.969,Z 237.343,A -85,B 0,C 180,E1 -4192.577,E2 -4192.577} C_VEL
LIN {X 0,Y 530.886,Z 237.356,A -85,B 0,C 180,E1 -4194.375,E2 -4194.375} C_VEL
LIN {X 0,Y 530.945,Z 238.262,A -85,B 0,C 180,E1 -4195.307,E2 -4195.307} C_VEL
LIN {X 0,Y 530.847,Z 242.417,A -85,B 0,C 180,E1 -4198.024,E2 -4198.024} C_VEL
LIN {X 0,Y 530.798,Z 246.926,A -85,B 0,C 180,E1 -4200.912,E2 -4200.912} C_VEL
LIN {X 0,Y 530.688,Z 250.627,A -85,B 0,C 180,E1 -4203.239,E2 -4203.239} C_VEL
LIN {X 0,Y 530.703,Z 255.141,A -85,B 0,C 180,E1 -4206.03,E2 -4206.03} C_VEL
LIN {X 0,Y 530.602,Z 260.147,A -85,B 0,C 180,E1 -4209.046,E2 -4209.046} C_VEL
LIN {X 0,Y 530.54,Z 264.231,A -85,B 0,C 180,E1 -4211.463,E2 -4211.463} C_VEL
LIN {X 0,Y 530.517,Z 268.32,A -85,B 0,C 180,E1 -4213.847,E2 -4213.847} C_VEL
LIN {X 0,Y 530.498,Z 272.427,A -85,B 0,C 180,E1 -4216.204,E2 -4216.204} C_VEL
LIN {X 0,Y 530.494,Z 273.018,A -85,B 0,C 180,E1 -4216.546,E2 -4216.546} C_VEL
LIN {X 0,Y 532.291,Z 283.663,A -85,B 0,C 180,E1 -4216.859,E2 -4216.859} C_VEL
LIN {X 0,Y 532.076,Z 296.609,A -85,B 0,C 180,E1 -4217.315,E2 -4217.315} C_VEL
LIN {X 0,Y 531.873,Z 308.838,A -85,B 0,C 180,E1 -4217.909,E2 -4217.909} C_VEL
LIN {X 0,Y 531.607,Z 320.67,A -85,B 0,C 180,E1 -4218.659,E2 -4218.659} C_VEL
LIN {X 0,Y 531.317,Z 331.37,A -85,B 0,C 180,E1 -4219.521,E2 -4219.521} C_VEL
LIN {X 0,Y 531.102,Z 340.995,A -85,B 0,C 180,E1 -4220.479,E2 -4220.479} C_VEL
LIN {X 0,Y 530.898,Z 348.878,A -85,B 0,C 180,E1 -4221.435,E2 -4221.435} C_VEL
LIN {X 0,Y 530.723,Z 356.588,A -85,B 0,C 180,E1 -4222.582,E2 -4222.582} C_VEL
LIN {X 0,Y 530.63,Z 363.656,A -85,B 0,C 180,E1 -4223.918,E2 -4223.918} C_VEL
LIN {X 0,Y 530.459,Z 368.37,A -85,B 0,C 180,E1 -4225.06,E2 -4225.06} C_VEL
LIN {X 0,Y 530.516,Z 371.977,A -85,B 0,C 180,E1 -4226.202,E2 -4226.202} C_VEL
LIN {X 0,Y 530.457,Z 373.844,A -85,B 0,C 180,E1 -4226.962,E2 -4226.962} C_VEL
LIN {X 0,Y 530.41,Z 375.253,A -85,B 0,C 180,E1 -4227.722,E2 -4227.722} C_VEL
LIN {X 0,Y 530.344,Z 376.873,A -85,B 0,C 180,E1 -4229.241,E2 -4229.241} C_VEL
LIN {X 0,Y 530.344,Z 377.111,A -85,B 0,C 180,E1 -4230,E2 -4230} C_VEL
LIN {X 0,Y 530.344,Z 376.929,A -85,B 0,C 180,E1 -4230.759,E2 -4230.759} C_VEL
LIN {X 0,Y 530.41,Z 375.382,A -85,B 0,C 180,E1 -4232.278,E2 -4232.278} C_VEL
LIN {X 0,Y 530.458,Z 374.028,A -85,B 0,C 180,E1 -4233.038,E2 -4233.038} C_VEL
LIN {X 0,Y 530.522,Z 371.167,A -85,B 0,C 180,E1 -4234.178,E2 -4234.178} C_VEL
LIN {X 0,Y 530.523,Z 367.289,A -85,B 0,C 180,E1 -4235.321,E2 -4235.321} C_VEL
LIN {X 0,Y 530.622,Z 361.591,A -85,B 0,C 180,E1 -4236.603,E2 -4236.603} C_VEL
LIN {X 0,Y 530.779,Z 354.76,A -85,B 0,C 180,E1 -4237.8,E2 -4237.8} C_VEL
LIN {X 0,Y 530.918,Z 346.615,A -85,B 0,C 180,E1 -4238.948,E2 -4238.948} C_VEL
LIN {X 0,Y 531.132,Z 338.276,A -85,B 0,C 180,E1 -4239.905,E2 -4239.905} C_VEL
LIN {X 0,Y 531.387,Z 327.983,A -85,B 0,C 180,E1 -4240.863,E2 -4240.863} C_VEL
LIN {X 0,Y 531.659,Z 317.456,A -85,B 0,C 180,E1 -4241.652,E2 -4241.652} C_VEL
LIN {X 0,Y 531.909,Z 306.629,A -85,B 0,C 180,E1 -4242.302,E2 -4242.302} C_VEL
LIN {X 0,Y 532.145,Z 294.108,A -85,B 0,C 180,E1 -4242.878,E2 -4242.878} C_VEL
LIN {X 0,Y 532.136,Z 282.038,A -85,B 0,C 180,E1 -4243.278,E2 -4243.278} C_VEL
LIN {X 0,Y 530.48,Z 272.947,A -85,B 0,C 180,E1 -4243.552,E2 -4243.552} C_VEL
LIN {X 0,Y 530.516,Z 269.832,A -85,B 0,C 180,E1 -4245.364,E2 -4245.364} C_VEL
LIN {X 0,Y 530.55,Z 265.771,A -85,B 0,C 180,E1 -4247.739,E2 -4247.739} C_VEL
LIN {X 0,Y 530.595,Z 261.659,A -85,B 0,C 180,E1 -4250.144,E2 -4250.144} C_VEL
LIN {X 0,Y 530.654,Z 257.579,A -85,B 0,C 180,E1 -4252.587,E2 -4252.587} C_VEL
LIN {X 0,Y 530.691,Z 253.491,A -85,B 0,C 180,E1 -4255.074,E2 -4255.074} C_VEL
LIN {X 0,Y 530.771,Z 248.049,A -85,B 0,C 180,E1 -4258.469,E2 -4258.469} C_VEL
LIN {X 0,Y 530.795,Z 243.947,A -85,B 0,C 180,E1 -4261.09,E2 -4261.09} C_VEL
LIN {X 0,Y 530.876,Z 239.798,A -85,B 0,C 180,E1 -4263.781,E2 -4263.781} C_VEL
LIN {X 0,Y 530.909,Z 238.186,A -85,B 0,C 180,E1 -4264.841,E2 -4264.841} C_VEL
LIN {X 0,Y 530.889,Z 237.356,A -85,B 0,C 180,E1 -4265.625,E2 -4265.625} C_VEL
LIN {X 0,Y 530.96,Z 237.348,A -85,B 0,C 180,E1 -4268.471,E2 -4268.471} C_VEL
LIN {X 0,Y 530.961,Z 237.344,A -85,B 0,C 180,E1 -4271.439,E2 -4271.439} C_VEL
LIN {X 0,Y 530.962,Z 237.345,A -85,B 0,C 180,E1 -4274.55,E2 -4274.55} C_VEL
LIN {X 0,Y 530.973,Z 237.344,A -85,B 0,C 180,E1 -4277.836,E2 -4277.836} C_VEL
LIN {X 0,Y 530.988,Z 237.347,A -85,B 0,C 180,E1 -4280.557,E2 -4280.557} C_VEL
LIN {X 0,Y 530.958,Z 237.344,A -85,B 0,C 180,E1 -4283.442,E2 -4283.442} C_VEL
LIN {X 0,Y 530.965,Z 237.344,A -85,B 0,C 180,E1 -4286.5,E2 -4286.5} C_VEL
LIN {X 0,Y 530.961,Z 237.35,A -85,B 0,C 180,E1 -4289.358,E2 -4289.358} C_VEL
LIN {X 0,Y 531.014,Z 237.343,A -85,B 0,C 180,E1 -4292.468,E2 -4292.468} C_VEL
LIN {X 0,Y 530.999,Z 237.34,A -85,B 0,C 180,E1 -4294.942,E2 -4294.942} C_VEL
LIN {X 0,Y 530.975,Z 237.343,A -85,B 0,C 180,E1 -4298.247,E2 -4298.247} C_VEL
LIN {X 0,Y 530.984,Z 237.341,A -85,B 0,C 180,E1 -4300.677,E2 -4300.677} C_VEL
LIN {X 0,Y 530.956,Z 237.35,A -85,B 0,C 180,E1 -4303.07,E2 -4303.07} C_VEL
LIN {X 0,Y 531.017,Z 237.338,A -85,B 0,C 180,E1 -4305.436,E2 -4305.436} C_VEL
LIN {X 0,Y 531.039,Z 237.336,A -85,B 0,C 180,E1 -4308.55,E2 -4308.55} C_VEL
LIN {X 0,Y 531.04,Z 237.338,A -85,B 0,C 180,E1 -4311.629,E2 -4311.629} C_VEL
LIN {X 0,Y 531.107,Z 237.329,A -85,B 0,C 180,E1 -4314.685,E2 -4314.685} C_VEL
LIN {X 0,Y 531.129,Z 237.324,A -85,B 0,C 180,E1 -4317.725,E2 -4317.725} C_VEL
LIN {X 0,Y 531.153,Z 237.321,A -85,B 0,C 180,E1 -4320.758,E2 -4320.758} C_VEL
LIN {X 0,Y 531.108,Z 237.328,A -85,B 0,C 180,E1 -4323.034,E2 -4323.034} C_VEL
LIN {X 0,Y 531.077,Z 237.33,A -85,B 0,C 180,E1 -4326.077,E2 -4326.077} C_VEL
LIN {X 0,Y 531.006,Z 237.338,A -85,B 0,C 180,E1 -4329.139,E2 -4329.139} C_VEL
LIN {X 0,Y 531.017,Z 237.342,A -85,B 0,C 180,E1 -4332.225,E2 -4332.225} C_VEL
LIN {X 0,Y 530.997,Z 237.344,A -85,B 0,C 180,E1 -4335.35,E2 -4335.35} C_VEL
LIN {X 0,Y 530.992,Z 237.343,A -85,B 0,C 180,E1 -4338.521,E2 -4338.521} C_VEL
LIN {X 0,Y 531.002,Z 237.342,A -85,B 0,C 180,E1 -4340.938,E2 -4340.938} C_VEL
LIN {X 0,Y 530.953,Z 237.348,A -85,B 0,C 180,E1 -4344.226,E2 -4344.226} C_VEL
LIN {X 0,Y 530.96,Z 237.344,A -85,B 0,C 180,E1 -4346.746,E2 -4346.746} C_VEL
LIN {X 0,Y 530.981,Z 237.347,A -85,B 0,C 180,E1 -4349.323,E2 -4349.323} C_VEL
LIN {X 0,Y 530.969,Z 237.345,A -85,B 0,C 180,E1 -4352.1,E2 -4352.1} C_VEL
LIN {X 0,Y 530.971,Z 237.344,A -85,B 0,C 180,E1 -4354.851,E2 -4354.851} C_VEL
LIN {X 0,Y 530.964,Z 237.348,A -85,B 0,C 180,E1 -4357.508,E2 -4357.508} C_VEL
LIN {X 0,Y 530.952,Z 237.345,A -85,B 0,C 180,E1 -4360.436,E2 -4360.436} C_VEL
LIN {X 0,Y 530.947,Z 237.347,A -85,B 0,C 180,E1 -4363.497,E2 -4363.497} C_VEL
LIN {X 0,Y 530.957,Z 237.349,A -85,B 0,C 180,E1 -4366.504,E2 -4366.504} C_VEL
LIN {X 0,Y 530.986,Z 237.343,A -85,B 0,C 180,E1 -4368.976,E2 -4368.976} C_VEL
LIN {X 0,Y 530.955,Z 237.351,A -85,B 0,C 180,E1 -4371.529,E2 -4371.529} C_VEL
LIN {X 0,Y 531.014,Z 237.454,A -85,B 0,C 180,E1 -4372.795,E2 -4372.795} C_VEL
LIN {X 0,Y 531.523,Z 241.123,A -85,B 0,C 180,E1 -4374.424,E2 -4374.424} C_VEL
LIN {X 0,Y 531.439,Z 247.726,A -85,B 0,C 180,E1 -4377.166,E2 -4377.166} C_VEL
LIN {X 0,Y 531.258,Z 255.523,A -85,B 0,C 180,E1 -4380.258,E2 -4380.258} C_VEL
LIN {X 0,Y 531.062,Z 263.372,A -85,B 0,C 180,E1 -4383.259,E2 -4383.259} C_VEL
LIN {X 0,Y 530.965,Z 270.634,A -85,B 0,C 180,E1 -4385.966,E2 -4385.966} C_VEL
LIN {X 0,Y 530.879,Z 277.979,A -85,B 0,C 180,E1 -4388.65,E2 -4388.65} C_VEL
LIN {X 0,Y 530.738,Z 285.766,A -85,B 0,C 180,E1 -4391.47,E2 -4391.47} C_VEL
LIN {X 0,Y 530.657,Z 293.717,A -85,B 0,C 180,E1 -4394.246,E2 -4394.246} C_VEL
LIN {X 0,Y 530.636,Z 300.401,A -85,B 0,C 180,E1 -4396.488,E2 -4396.488} C_VEL
LIN {X 0,Y 532.313,Z 310.877,A -85,B 0,C 180,E1 -4396.763,E2 -4396.763} C_VEL
LIN {X 0,Y 532.116,Z 323.407,A -85,B 0,C 180,E1 -4397.17,E2 -4397.17} C_VEL
LIN {X 0,Y 531.85,Z 335.063,A -85,B 0,C 180,E1 -4397.697,E2 -4397.697} C_VEL
LIN {X 0,Y 531.598,Z 346.276,A -85,B 0,C 180,E1 -4398.358,E2 -4398.358} C_VEL
LIN {X 0,Y 531.347,Z 357.99,A -85,B 0,C 180,E1 -4399.232,E2 -4399.232} C_VEL
LIN {X 0,Y 531.098,Z 367.3,A -85,B 0,C 180,E1 -4400.094,E2 -4400.094} C_VEL
LIN {X 0,Y 530.931,Z 375.79,A -85,B 0,C 180,E1 -4401.052,E2 -4401.052} C_VEL
LIN {X 0,Y 530.734,Z 384.071,A -85,B 0,C 180,E1 -4402.199,E2 -4402.199} C_VEL
LIN {X 0,Y 530.598,Z 391.142,A -85,B 0,C 180,E1 -4403.419,E2 -4403.419} C_VEL
LIN {X 0,Y 530.524,Z 396.856,A -85,B 0,C 180,E1 -4404.679,E2 -4404.679} C_VEL
LIN {X 0,Y 530.522,Z 400.825,A -85,B 0,C 180,E1 -4405.822,E2 -4405.822} C_VEL
LIN {X 0,Y 530.457,Z 403.755,A -85,B 0,C 180,E1 -4406.962,E2 -4406.962} C_VEL
LIN {X 0,Y 530.411,Z 405.149,A -85,B 0,C 180,E1 -4407.722,E2 -4407.722} C_VEL
LIN {X 0,Y 530.344,Z 406.75,A -85,B 0,C 180,E1 -4409.241,E2 -4409.241} C_VEL
LIN {X 0,Y 530.343,Z 406.967,A -85,B 0,C 180,E1 -4410,E2 -4410} C_VEL
LIN {X 0,Y 530.361,Z 406.145,A -85,B 0,C 180,E1 -4411.519,E2 -4411.519} C_VEL
LIN {X 0,Y 530.411,Z 405.152,A -85,B 0,C 180,E1 -4412.278,E2 -4412.278} C_VEL
LIN {X 0,Y 530.457,Z 403.759,A -85,B 0,C 180,E1 -4413.038,E2 -4413.038} C_VEL
LIN {X 0,Y 530.522,Z 400.827,A -85,B 0,C 180,E1 -4414.178,E2 -4414.178} C_VEL
LIN {X 0,Y 530.524,Z 396.855,A -85,B 0,C 180,E1 -4415.321,E2 -4415.321} C_VEL
LIN {X 0,Y 530.596,Z 391.152,A -85,B 0,C 180,E1 -4416.579,E2 -4416.579} C_VEL
LIN {X 0,Y 530.734,Z 384.073,A -85,B 0,C 180,E1 -4417.801,E2 -4417.801} C_VEL
LIN {X 0,Y 530.931,Z 375.791,A -85,B 0,C 180,E1 -4418.948,E2 -4418.948} C_VEL
LIN {X 0,Y 531.098,Z 367.302,A -85,B 0,C 180,E1 -4419.906,E2 -4419.906} C_VEL
LIN {X 0,Y 531.359,Z 356.814,A -85,B 0,C 180,E1 -4420.864,E2 -4420.864} C_VEL
LIN {X 0,Y 531.645,Z 344.994,A -85,B 0,C 180,E1 -4421.728,E2 -4421.728} C_VEL
LIN {X 0,Y 531.88,Z 333.14,A -85,B 0,C 180,E1 -4422.399,E2 -4422.399} C_VEL
LIN {X 0,Y 532.166,Z 320.795,A -85,B 0,C 180,E1 -4422.925,E2 -4422.925} C_VEL
LIN {X 0,Y 532.122,Z 309.496,A -85,B 0,C 180,E1 -4423.279,E2 -4423.279} C_VEL
LIN {X 0,Y 530.606,Z 300.158,A -85,B 0,C 180,E1 -4423.524,E2 -4423.524} C_VEL
LIN {X 0,Y 530.688,Z 291.449,A -85,B 0,C 180,E1 -4426.543,E2 -4426.543} C_VEL
LIN {X 0,Y 530.788,Z 283.544,A -85,B 0,C 180,E1 -4429.331,E2 -4429.331} C_VEL
LIN {X 0,Y 530.913,Z 275.956,A -85,B 0,C 180,E1 -4432.084,E2 -4432.084} C_VEL
LIN {X 0,Y 531.007,Z 267.865,A -85,B 0,C 180,E1 -4435.057,E2 -4435.057} C_VEL
LIN {X 0,Y 531.12,Z 260.002,A -85,B 0,C 180,E1 -4438.018,E2 -4438.018} C_VEL
LIN {X 0,Y 531.28,Z 253.071,A -85,B 0,C 180,E1 -4440.7,E2 -4440.7} C_VEL
LIN {X 0,Y 531.438,Z 247.715,A -85,B 0,C 180,E1 -4442.834,E2 -4442.834} C_VEL
LIN {X 0,Y 531.522,Z 241.113,A -85,B 0,C 180,E1 -4445.576,E2 -4445.576} C_VEL
LIN {X 0,Y 530.959,Z 237.35,A -85,B 0,C 180,E1 -4447.281,E2 -4447.281} C_VEL
LIN {X 0,Y 530.983,Z 237.349,A -85,B 0,C 180,E1 -4450.433,E2 -4450.433} C_VEL
LIN {X 0,Y 530.963,Z 237.346,A -85,B 0,C 180,E1 -4453.281,E2 -4453.281} C_VEL
LIN {X 0,Y 530.978,Z 237.346,A -85,B 0,C 180,E1 -4455.622,E2 -4455.622} C_VEL
LIN {X 0,Y 530.964,Z 237.347,A -85,B 0,C 180,E1 -4458.561,E2 -4458.561} C_VEL
LIN {X 0,Y 530.95,Z 237.345,A -85,B 0,C 180,E1 -4461.529,E2 -4461.529} C_VEL
LIN {X 0,Y 530.952,Z 237.348,A -85,B 0,C 180,E1 -4464.38,E2 -4464.38} C_VEL
LIN {X 0,Y 530.972,Z 237.346,A -85,B 0,C 180,E1 -4467.134,E2 -4467.134} C_VEL
LIN {X 0,Y 530.97,Z 237.344,A -85,B 0,C 180,E1 -4469.803,E2 -4469.803} C_VEL
LIN {X 0,Y 530.968,Z 237.349,A -85,B 0,C 180,E1 -4472.477,E2 -4472.477} C_VEL
LIN {X 0,Y 530.951,Z 237.345,A -85,B 0,C 180,E1 -4474.94,E2 -4474.94} C_VEL
LIN {X 0,Y 530.979,Z 237.346,A -85,B 0,C 180,E1 -4477.898,E2 -4477.898} C_VEL
LIN {X 0,Y 530.995,Z 237.342,A -85,B 0,C 180,E1 -4480.677,E2 -4480.677} C_VEL
LIN {X 0,Y 530.986,Z 237.346,A -85,B 0,C 180,E1 -4483.071,E2 -4483.071} C_VEL
LIN {X 0,Y 531.018,Z 237.338,A -85,B 0,C 180,E1 -4485.436,E2 -4485.436} C_VEL
LIN {X 0,Y 531.033,Z 237.336,A -85,B 0,C 180,E1 -4488.55,E2 -4488.55} C_VEL
LIN {X 0,Y 531.03,Z 237.339,A -85,B 0,C 180,E1 -4491.629,E2 -4491.629} C_VEL
LIN {X 0,Y 531.076,Z 237.33,A -85,B 0,C 180,E1 -4493.923,E2 -4493.923} C_VEL
LIN {X 0,Y 531.107,Z 237.329,A -85,B 0,C 180,E1 -4496.966,E2 -4496.966} C_VEL
LIN {X 0,Y 531.145,Z 237.326,A -85,B 0,C 180,E1 -4500,E2 -4500} C_VEL
LIN {X 0,Y 531.09,Z 237.33,A -85,B 0,C 180,E1 -4503.034,E2 -4503.034} C_VEL
LIN {X 0,Y 531.049,Z 237.332,A -85,B 0,C 180,E1 -4506.078,E2 -4506.078} C_VEL
LIN {X 0,Y 531.028,Z 237.337,A -85,B 0,C 180,E1 -4509.138,E2 -4509.138} C_VEL
LIN {X 0,Y 531.042,Z 237.339,A -85,B 0,C 180,E1 -4512.225,E2 -4512.225} C_VEL
LIN {X 0,Y 530.988,Z 237.346,A -85,B 0,C 180,E1 -4515.35,E2 -4515.35} C_VEL
LIN {X 0,Y 530.973,Z 237.345,A -85,B 0,C 180,E1 -4518.522,E2 -4518.522} C_VEL
LIN {X 0,Y 531,Z 237.34,A -85,B 0,C 180,E1 -4520.938,E2 -4520.938} C_VEL
LIN {X 0,Y 530.968,Z 237.347,A -85,B 0,C 180,E1 -4524.225,E2 -4524.225} C_VEL
LIN {X 0,Y 531.003,Z 237.34,A -85,B 0,C 180,E1 -4526.744,E2 -4526.744} C_VEL
LIN {X 0,Y 530.979,Z 237.346,A -85,B 0,C 180,E1 -4529.323,E2 -4529.323} C_VEL
LIN {X 0,Y 530.965,Z 237.345,A -85,B 0,C 180,E1 -4532.1,E2 -4532.1} C_VEL
LIN {X 0,Y 530.965,Z 237.343,A -85,B 0,C 180,E1 -4534.85,E2 -4534.85} C_VEL
LIN {X 0,Y 530.965,Z 237.347,A -85,B 0,C 180,E1 -4537.508,E2 -4537.508} C_VEL
LIN {X 0,Y 530.983,Z 237.342,A -85,B 0,C 180,E1 -4540.433,E2 -4540.433} C_VEL
LIN {X 0,Y 530.935,Z 237.35,A -85,B 0,C 180,E1 -4543.278,E2 -4543.278} C_VEL
LIN {X 0,Y 530.937,Z 237.348,A -85,B 0,C 180,E1 -4543.545,E2 -4543.545} C_VEL
LIN {X 0,Y 530.268,Z 237.435,A -85,B 0,C 180,E1 -4544.179,E2 -4544.179} C_VEL
LIN {X 0,Y 527.422,Z 237.787,A -85,B 0,C 180,E1 -4545.207,E2 -4545.207} C_VEL
LIN {X 0,Y 525.012,Z 238.09,A -85,B 0,C 180,E1 -4546.036,E2 -4546.036} C_VEL
LIN {X 0,Y 523.968,Z 238.217,A -85,B 0,C 180,E1 -4546.675,E2 -4546.675} C_VEL
LIN {X 0,Y 523.877,Z 238.227,A -85,B 0,C 180,E1 -4546.892,E2 -4546.892} C_VEL
LIN {X 0,Y 523.915,Z 238.224,A -85,B 0,C 180,E1 -4549.917,E2 -4549.917} C_VEL
LIN {X 0,Y 523.905,Z 238.227,A -85,B 0,C 180,E1 -4552.868,E2 -4552.868} C_VEL
LIN {X 0,Y 523.83,Z 238.324,A -85,B 0,C 180,E1 -4554.766,E2 -4554.766} C_VEL
LIN {X 0,Y 523.814,Z 242.499,A -85,B 0,C 180,E1 -4557.542,E2 -4557.542} C_VEL
LIN {X 0,Y 523.734,Z 247.389,A -85,B 0,C 180,E1 -4560.72,E2 -4560.72} C_VEL
LIN {X 0,Y 523.636,Z 252.094,A -85,B 0,C 180,E1 -4563.71,E2 -4563.71} C_VEL
LIN {X 0,Y 523.629,Z 256.174,A -85,B 0,C 180,E1 -4566.256,E2 -4566.256} C_VEL
LIN {X 0,Y 523.532,Z 260.263,A -85,B 0,C 180,E1 -4568.749,E2 -4568.749} C_VEL
LIN {X 0,Y 523.481,Z 264.369,A -85,B 0,C 180,E1 -4571.203,E2 -4571.203} C_VEL
LIN {X 0,Y 523.439,Z 268.478,A -85,B 0,C 180,E1 -4573.623,E2 -4573.623} C_VEL
LIN {X 0,Y 523.444,Z 272.632,A -85,B 0,C 180,E1 -4576.015,E2 -4576.015} C_VEL
LIN {X 0,Y 523.424,Z 273.281,A -85,B 0,C 180,E1 -4576.373,E2 -4576.373} C_VEL
LIN {X 0,Y 525.396,Z 284.698,A -85,B 0,C 180,E1 -4576.708,E2 -4576.708} C_VEL
LIN {X 0,Y 525.151,Z 297.95,A -85,B 0,C 180,E1 -4577.194,E2 -4577.194} C_VEL
LIN {X 0,Y 524.936,Z 309.691,A -85,B 0,C 180,E1 -4577.782,E2 -4577.782} C_VEL
LIN {X 0,Y 524.652,Z 320.878,A -85,B 0,C 180,E1 -4578.506,E2 -4578.506} C_VEL
LIN {X 0,Y 524.339,Z 331.576,A -85,B 0,C 180,E1 -4579.38,E2 -4579.38} C_VEL
LIN {X 0,Y 524.081,Z 341.201,A -85,B 0,C 180,E1 -4580.35,E2 -4580.35} C_VEL
LIN {X 0,Y 523.873,Z 349.083,A -85,B 0,C 180,E1 -4581.32,E2 -4581.32} C_VEL
LIN {X 0,Y 523.663,Z 356.792,A -85,B 0,C 180,E1 -4582.481,E2 -4582.481} C_VEL
LIN {X 0,Y 523.565,Z 363.858,A -85,B 0,C 180,E1 -4583.835,E2 -4583.835} C_VEL
LIN {X 0,Y 523.384,Z 368.573,A -85,B 0,C 180,E1 -4584.993,E2 -4584.993} C_VEL
LIN {X 0,Y 523.443,Z 372.178,A -85,B 0,C 180,E1 -4586.151,E2 -4586.151} C_VEL
LIN {X 0,Y 523.367,Z 374.045,A -85,B 0,C 180,E1 -4586.921,E2 -4586.921} C_VEL
LIN {X 0,Y 523.334,Z 375.453,A -85,B 0,C 180,E1 -4587.691,E2 -4587.691} C_VEL
LIN {X 0,Y 523.25,Z 377.073,A -85,B 0,C 180,E1 -4589.23,E2 -4589.23} C_VEL
LIN {X 0,Y 523.247,Z 377.311,A -85,B 0,C 180,E1 -4590,E2 -4590} C_VEL
LIN {X 0,Y 523.25,Z 377.128,A -85,B 0,C 180,E1 -4590.77,E2 -4590.77} C_VEL
LIN {X 0,Y 523.334,Z 375.581,A -85,B 0,C 180,E1 -4592.309,E2 -4592.309} C_VEL
LIN {X 0,Y 523.368,Z 374.227,A -85,B 0,C 180,E1 -4593.079,E2 -4593.079} C_VEL
LIN {X 0,Y 523.442,Z 371.365,A -85,B 0,C 180,E1 -4594.235,E2 -4594.235} C_VEL
LIN {X 0,Y 523.463,Z 367.486,A -85,B 0,C 180,E1 -4595.393,E2 -4595.393} C_VEL
LIN {X 0,Y 523.571,Z 362.127,A -85,B 0,C 180,E1 -4596.625,E2 -4596.625} C_VEL
LIN {X 0,Y 523.728,Z 354.956,A -85,B 0,C 180,E1 -4597.906,E2 -4597.906} C_VEL
LIN {X 0,Y 523.898,Z 346.81,A -85,B 0,C 180,E1 -4599.069,E2 -4599.069} C_VEL
LIN {X 0,Y 524.128,Z 338.471,A -85,B 0,C 180,E1 -4600.039,E2 -4600.039} C_VEL
LIN {X 0,Y 524.416,Z 328.176,A -85,B 0,C 180,E1 -4601.01,E2 -4601.01} C_VEL
LIN {X 0,Y 524.747,Z 316.767,A -85,B 0,C 180,E1 -4601.869,E2 -4601.869} C_VEL
LIN {X 0,Y 525.03,Z 305.005,A -85,B 0,C 180,E1 -4602.564,E2 -4602.564} C_VEL
LIN {X 0,Y 525.272,Z 292.992,A -85,B 0,C 180,E1 -4603.098,E2 -4603.098} C_VEL
LIN {X 0,Y 525.247,Z 283.128,A -85,B 0,C 180,E1 -4603.431,E2 -4603.431} C_VEL
LIN {X 0,Y 523.426,Z 273.15,A -85,B 0,C 180,E1 -4603.738,E2 -4603.738} C_VEL
LIN {X 0,Y 523.429,Z 269.996,A -85,B 0,C 180,E1 -4605.577,E2 -4605.577} C_VEL
LIN {X 0,Y 523.457,Z 265.897,A -85,B 0,C 180,E1 -4607.987,E2 -4607.987} C_VEL
LIN {X 0,Y 523.517,Z 261.773,A -85,B 0,C 180,E1 -4610.429,E2 -4610.429} C_VEL
LIN {X 0,Y 523.578,Z 257.681,A -85,B 0,C 180,E1 -4612.909,E2 -4612.909} C_VEL
LIN {X 0,Y 523.625,Z 253.602,A -85,B 0,C 180,E1 -4615.436,E2 -4615.436} C_VEL
LIN {X 0,Y 523.69,Z 249.513,A -85,B 0,C 180,E1 -4618.015,E2 -4618.015} C_VEL
LIN {X 0,Y 523.73,Z 245.172,A -85,B 0,C 180,E1 -4620.815,E2 -4620.815} C_VEL
LIN {X 0,Y 523.829,Z 240.746,A -85,B 0,C 180,E1 -4623.713,E2 -4623.713} C_VEL
LIN {X 0,Y 523.824,Z 238.466,A -85,B 0,C 180,E1 -4625.234,E2 -4625.234} C_VEL
LIN {X 0,Y 523.911,Z 238.222,A -85,B 0,C 180,E1 -4627.678,E2 -4627.678} C_VEL
LIN {X 0,Y 523.941,Z 238.221,A -85,B 0,C 180,E1 -4630.13,E2 -4630.13} C_VEL
LIN {X 0,Y 523.882,Z 238.227,A -85,B 0,C 180,E1 -4633.171,E2 -4633.171} C_VEL
LIN {X 0,Y 523.925,Z 238.225,A -85,B 0,C 180,E1 -4635.77,E2 -4635.77} C_VEL
LIN {X 0,Y 523.94,Z 238.223,A -85,B 0,C 180,E1 -4638.908,E2 -4638.908} C_VEL
LIN {X 0,Y 523.918,Z 238.223,A -85,B 0,C 180,E1 -4641.898,E2 -4641.898} C_VEL
LIN {X 0,Y 523.926,Z 238.219,A -85,B 0,C 180,E1 -4644.911,E2 -4644.911} C_VEL
LIN {X 0,Y 523.937,Z 238.224,A -85,B 0,C 180,E1 -4647.68,E2 -4647.68} C_VEL
LIN {X 0,Y 523.954,Z 238.221,A -85,B 0,C 180,E1 -4650.677,E2 -4650.677} C_VEL
LIN {X 0,Y 523.977,Z 238.215,A -85,B 0,C 180,E1 -4653.729,E2 -4653.729} C_VEL
LIN {X 0,Y 523.916,Z 238.225,A -85,B 0,C 180,E1 -4656.27,E2 -4656.27} C_VEL
LIN {X 0,Y 523.949,Z 238.217,A -85,B 0,C 180,E1 -4658.767,E2 -4658.767} C_VEL
LIN {X 0,Y 523.938,Z 238.224,A -85,B 0,C 180,E1 -4661.22,E2 -4661.22} C_VEL
LIN {X 0,Y 523.894,Z 238.225,A -85,B 0,C 180,E1 -4663.637,E2 -4663.637} C_VEL
LIN {X 0,Y 523.932,Z 238.223,A -85,B 0,C 180,E1 -4666.028,E2 -4666.028} C_VEL
LIN {X 0,Y 524.017,Z 238.213,A -85,B 0,C 180,E1 -4668.394,E2 -4668.394} C_VEL
LIN {X 0,Y 523.993,Z 238.217,A -85,B 0,C 180,E1 -4671.516,E2 -4671.516} C_VEL
LIN {X 0,Y 524.017,Z 238.208,A -85,B 0,C 180,E1 -4673.841,E2 -4673.841} C_VEL
LIN {X 0,Y 524.033,Z 238.21,A -85,B 0,C 180,E1 -4676.925,E2 -4676.925} C_VEL
LIN {X 0,Y 523.996,Z 238.218,A -85,B 0,C 180,E1 -4678.463,E2 -4678.463} C_VEL
LIN {X 0,Y 524.124,Z 238.197,A -85,B 0,C 180,E1 -4680.768,E2 -4680.768} C_VEL
LIN {X 0,Y 524.074,Z 238.205,A -85,B 0,C 180,E1 -4683.075,E2 -4683.075} C_VEL
LIN {X 0,Y 524.039,Z 238.207,A -85,B 0,C 180,E1 -4686.159,E2 -4686.159} C_VEL
LIN {X 0,Y 523.983,Z 238.218,A -85,B 0,C 180,E1 -4688.484,E2 -4688.484} C_VEL
LIN {X 0,Y 523.977,Z 238.216,A -85,B 0,C 180,E1 -4691.724,E2 -4691.724} C_VEL
LIN {X 0,Y 523.995,Z 238.214,A -85,B 0,C 180,E1 -4695.052,E2 -4695.052} C_VEL
LIN {X 0,Y 523.967,Z 238.216,A -85,B 0,C 180,E1 -4697.969,E2 -4697.969} C_VEL
LIN {X 0,Y 523.975,Z 238.219,A -85,B 0,C 180,E1 -4700.41,E2 -4700.41} C_VEL
LIN {X 0,Y 523.911,Z 238.222,A -85,B 0,C 180,E1 -4702.894,E2 -4702.894} C_VEL
LIN {X 0,Y 523.901,Z 238.225,A -85,B 0,C 180,E1 -4705.421,E2 -4705.421} C_VEL
LIN {X 0,Y 523.918,Z 238.223,A -85,B 0,C 180,E1 -4708.002,E2 -4708.002} C_VEL
LIN {X 0,Y 523.939,Z 238.223,A -85,B 0,C 180,E1 -4710.853,E2 -4710.853} C_VEL
LIN {X 0,Y 523.962,Z 238.218,A -85,B 0,C 180,E1 -4713.734,E2 -4713.734} C_VEL
LIN {X 0,Y 523.901,Z 238.226,A -85,B 0,C 180,E1 -4716.4,E2 -4716.4} C_VEL
LIN {X 0,Y 523.912,Z 238.224,A -85,B 0,C 180,E1 -4719.086,E2 -4719.086} C_VEL
LIN {X 0,Y 523.914,Z 238.222,A -85,B 0,C 180,E1 -4722.123,E2 -4722.123} C_VEL
LIN {X 0,Y 523.945,Z 238.219,A -85,B 0,C 180,E1 -4725.31,E2 -4725.31} C_VEL
LIN {X 0,Y 523.958,Z 238.218,A -85,B 0,C 180,E1 -4728.69,E2 -4728.69} C_VEL
LIN {X 0,Y 523.919,Z 238.226,A -85,B 0,C 180,E1 -4731.898,E2 -4731.898} C_VEL
LIN {X 0,Y 524.003,Z 238.445,A -85,B 0,C 180,E1 -4732.671,E2 -4732.671} C_VEL
LIN {X 0,Y 524.535,Z 243.248,A -85,B 0,C 180,E1 -4734.82,E2 -4734.82} C_VEL
LIN {X 0,Y 524.419,Z 249.908,A -85,B 0,C 180,E1 -4737.597,E2 -4737.597} C_VEL
LIN {X 0,Y 524.226,Z 257.473,A -85,B 0,C 180,E1 -4740.624,E2 -4740.624} C_VEL
LIN {X 0,Y 524.006,Z 266.161,A -85,B 0,C 180,E1 -4743.976,E2 -4743.976} C_VEL
LIN {X 0,Y 523.859,Z 274.497,A -85,B 0,C 180,E1 -4747.104,E2 -4747.104} C_VEL
LIN {X 0,Y 523.752,Z 282.192,A -85,B 0,C 180,E1 -4749.935,E2 -4749.935} C_VEL
LIN {X 0,Y 523.63,Z 290.155,A -85,B 0,C 180,E1 -4752.826,E2 -4752.826} C_VEL
LIN {X 0,Y 523.55,Z 299.225,A -85,B 0,C 180,E1 -4756.017,E2 -4756.017} C_VEL
LIN {X 0,Y 523.543,Z 300.196,A -85,B 0,C 180,E1 -4756.302,E2 -4756.302} C_VEL
LIN {X 0,Y 525.354,Z 311.593,A -85,B 0,C 180,E1 -4756.609,E2 -4756.609} C_VEL
LIN {X 0,Y 525.152,Z 324.415,A -85,B 0,C 180,E1 -4757.046,E2 -4757.046} C_VEL
LIN {X 0,Y 524.861,Z 336.632,A -85,B 0,C 180,E1 -4757.629,E2 -4757.629} C_VEL
LIN {X 0,Y 524.546,Z 348.063,A -85,B 0,C 180,E1 -4758.336,E2 -4758.336} C_VEL
LIN {X 0,Y 524.326,Z 358.927,A -85,B 0,C 180,E1 -4759.184,E2 -4759.184} C_VEL
LIN {X 0,Y 524.036,Z 368.9,A -85,B 0,C 180,E1 -4760.154,E2 -4760.154} C_VEL
LIN {X 0,Y 523.821,Z 378.572,A -85,B 0,C 180,E1 -4761.319,E2 -4761.319} C_VEL
LIN {X 0,Y 523.629,Z 386.27,A -85,B 0,C 180,E1 -4762.481,E2 -4762.481} C_VEL
LIN {X 0,Y 523.494,Z 393.366,A -85,B 0,C 180,E1 -4763.834,E2 -4763.834} C_VEL
LIN {X 0,Y 523.383,Z 398.086,A -85,B 0,C 180,E1 -4764.993,E2 -4764.993} C_VEL
LIN {X 0,Y 523.443,Z 401.696,A -85,B 0,C 180,E1 -4766.151,E2 -4766.151} C_VEL
LIN {X 0,Y 523.367,Z 403.555,A -85,B 0,C 180,E1 -4766.921,E2 -4766.921} C_VEL
LIN {X 0,Y 523.335,Z 404.949,A -85,B 0,C 180,E1 -4767.691,E2 -4767.691} C_VEL
LIN {X 0,Y 523.25,Z 406.551,A -85,B 0,C 180,E1 -4769.23,E2 -4769.23} C_VEL
LIN {X 0,Y 523.246,Z 406.767,A -85,B 0,C 180,E1 -4770,E2 -4770} C_VEL
LIN {X 0,Y 523.275,Z 405.945,A -85,B 0,C 180,E1 -4771.539,E2 -4771.539} C_VEL
LIN {X 0,Y 523.335,Z 404.953,A -85,B 0,C 180,E1 -4772.309,E2 -4772.309} C_VEL
LIN {X 0,Y 523.367,Z 403.559,A -85,B 0,C 180,E1 -4773.079,E2 -4773.079} C_VEL
LIN {X 0,Y 523.424,Z 400.626,A -85,B 0,C 180,E1 -4774.235,E2 -4774.235} C_VEL
LIN {X 0,Y 523.461,Z 396.655,A -85,B 0,C 180,E1 -4775.393,E2 -4775.393} C_VEL
LIN {X 0,Y 523.517,Z 391.431,A -85,B 0,C 180,E1 -4776.575,E2 -4776.575} C_VEL
LIN {X 0,Y 523.652,Z 385.109,A -85,B 0,C 180,E1 -4777.713,E2 -4777.713} C_VEL
LIN {X 0,Y 523.837,Z 377.082,A -85,B 0,C 180,E1 -4778.875,E2 -4778.875} C_VEL
LIN {X 0,Y 524.036,Z 368.902,A -85,B 0,C 180,E1 -4779.846,E2 -4779.846} C_VEL
LIN {X 0,Y 524.325,Z 358.928,A -85,B 0,C 180,E1 -4780.816,E2 -4780.816} C_VEL
LIN {X 0,Y 524.612,Z 347.737,A -85,B 0,C 180,E1 -4781.686,E2 -4781.686} C_VEL
LIN {X 0,Y 524.838,Z 336.634,A -85,B 0,C 180,E1 -4782.372,E2 -4782.372} C_VEL
LIN {X 0,Y 525.127,Z 324.409,A -85,B 0,C 180,E1 -4782.954,E2 -4782.954} C_VEL
LIN {X 0,Y 525.354,Z 311.59,A -85,B 0,C 180,E1 -4783.391,E2 -4783.391} C_VEL
LIN {X 0,Y 523.549,Z 300.004,A -85,B 0,C 180,E1 -4783.71,E2 -4783.71} C_VEL
LIN {X 0,Y 523.633,Z 291.293,A -85,B 0,C 180,E1 -4786.772,E2 -4786.772} C_VEL
LIN {X 0,Y 523.747,Z 283.449,A -85,B 0,C 180,E1 -4789.601,E2 -4789.601} C_VEL
LIN {X 0,Y 523.857,Z 276.306,A -85,B 0,C 180,E1 -4792.226,E2 -4792.226} C_VEL
LIN {X 0,Y 523.951,Z 268.88,A -85,B 0,C 180,E1 -4794.994,E2 -4794.994} C_VEL
LIN {X 0,Y 524.084,Z 261.026,A -85,B 0,C 180,E1 -4797.992,E2 -4797.992} C_VEL
LIN {X 0,Y 524.245,Z 254.316,A -85,B 0,C 180,E1 -4800.626,E2 -4800.626} C_VEL
LIN {X 0,Y 524.46,Z 247.652,A -85,B 0,C 180,E1 -4803.327,E2 -4803.327} C_VEL
LIN {X 0,Y 524.526,Z 242.154,A -85,B 0,C 180,E1 -4805.651,E2 -4805.651} C_VEL
LIN {X 0,Y 523.941,Z 238.224,A -85,B 0,C 180,E1 -4807.434,E2 -4807.434} C_VEL
LIN {X 0,Y 523.939,Z 238.225,A -85,B 0,C 180,E1 -4810.13,E2 -4810.13} C_VEL
LIN {X 0,Y 523.938,Z 238.221,A -85,B 0,C 180,E1 -4812.459,E2 -4812.459} C_VEL
LIN {X 0,Y 523.945,Z 238.224,A -85,B 0,C 180,E1 -4815.31,E2 -4815.31} C_VEL
LIN {X 0,Y 523.924,Z 238.225,A -85,B 0,C 180,E1 -4818.694,E2 -4818.694} C_VEL
LIN {X 0,Y 523.911,Z 238.223,A -85,B 0,C 180,E1 -4821.898,E2 -4821.898} C_VEL
LIN {X 0,Y 523.925,Z 238.221,A -85,B 0,C 180,E1 -4824.911,E2 -4824.911} C_VEL
LIN {X 0,Y 523.94,Z 238.223,A -85,B 0,C 180,E1 -4827.679,E2 -4827.679} C_VEL
LIN {X 0,Y 523.954,Z 238.222,A -85,B 0,C 180,E1 -4830.677,E2 -4830.677} C_VEL
LIN {X 0,Y 523.904,Z 238.224,A -85,B 0,C 180,E1 -4833.725,E2 -4833.725} C_VEL
LIN {X 0,Y 523.91,Z 238.225,A -85,B 0,C 180,E1 -4836.269,E2 -4836.269} C_VEL
LIN {X 0,Y 523.948,Z 238.218,A -85,B 0,C 180,E1 -4838.767,E2 -4838.767} C_VEL
LIN {X 0,Y 523.952,Z 238.222,A -85,B 0,C 180,E1 -4841.221,E2 -4841.221} C_VEL
LIN {X 0,Y 523.936,Z 238.22,A -85,B 0,C 180,E1 -4843.639,E2 -4843.639} C_VEL
LIN {X 0,Y 523.932,Z 238.224,A -85,B 0,C 180,E1 -4846.028,E2 -4846.028} C_VEL
LIN {X 0,Y 524.015,Z 238.211,A -85,B 0,C 180,E1 -4848.394,E2 -4848.394} C_VEL
LIN {X 0,Y 523.982,Z 238.219,A -85,B 0,C 180,E1 -4851.516,E2 -4851.516} C_VEL
LIN {X 0,Y 524.038,Z 238.207,A -85,B 0,C 180,E1 -4853.841,E2 -4853.841} C_VEL
LIN {X 0,Y 524.073,Z 238.205,A -85,B 0,C 180,E1 -4856.925,E2 -4856.925} C_VEL
LIN {X 0,Y 524.116,Z 238.201,A -85,B 0,C 180,E1 -4860,E2 -4860} C_VEL
LIN {X 0,Y 524.032,Z 238.21,A -85,B 0,C 180,E1 -4863.075,E2 -4863.075} C_VEL
LIN {X 0,Y 524.016,Z 238.208,A -85,B 0,C 180,E1 -4866.159,E2 -4866.159} C_VEL
LIN {X 0,Y 523.997,Z 238.212,A -85,B 0,C 180,E1 -4869.262,E2 -4869.262} C_VEL
LIN {X 0,Y 524.005,Z 238.215,A -85,B 0,C 180,E1 -4871.739,E2 -4871.739} C_VEL
LIN {X 0,Y 523.994,Z 238.215,A -85,B 0,C 180,E1 -4875.051,E2 -4875.051} C_VEL
LIN {X 0,Y 523.946,Z 238.218,A -85,B 0,C 180,E1 -4877.97,E2 -4877.97} C_VEL
LIN {X 0,Y 523.974,Z 238.219,A -85,B 0,C 180,E1 -4880.41,E2 -4880.41} C_VEL
LIN {X 0,Y 523.913,Z 238.222,A -85,B 0,C 180,E1 -4882.894,E2 -4882.894} C_VEL
LIN {X 0,Y 523.987,Z 238.216,A -85,B 0,C 180,E1 -4886.02,E2 -4886.02} C_VEL
LIN {X 0,Y 523.93,Z 238.224,A -85,B 0,C 180,E1 -4888.875,E2 -4888.875} C_VEL
LIN {X 0,Y 523.919,Z 238.222,A -85,B 0,C 180,E1 -4891.544,E2 -4891.544} C_VEL
LIN {X 0,Y 523.919,Z 238.227,A -85,B 0,C 180,E1 -4894.291,E2 -4894.291} C_VEL
LIN {X 0,Y 523.906,Z 238.223,A -85,B 0,C 180,E1 -4897.133,E2 -4897.133} C_VEL
LIN {X 0,Y 523.94,Z 238.219,A -85,B 0,C 180,E1 -4900.13,E2 -4900.13} C_VEL
LIN {X 0,Y 523.92,Z 238.224,A -85,B 0,C 180,E1 -4902.457,E2 -4902.457} C_VEL
LIN {X 0,Y 523.933,Z 238.22,A -85,B 0,C 180,E1 -4905.312,E2 -4905.312} C_VEL
